LIN {X 0,Y 486.099,Z 588.304,A -85,B 0,C 180,E1 16517.76,E2 16517.76} C_VEL
LIN {X 0,Y 480.059,Z 803.394,A -85,B 0,C 180,E1 16513.95,E2 16513.95} C_VEL
LIN {X 0,Y 477.626,Z 893.821,A -85,B 0,C 180,E1 16512.362,E2 16512.362} C_VEL
LIN {X 0,Y 476.267,Z 916.596,A -85,B 0,C 180,E1 16511.765,E2 16511.765} C_VEL
LIN {X 0,Y 474.605,Z 939.076,A -85,B 0,C 180,E1 16510.978,E2 16510.978} C_VEL
LIN {X 0,Y 472.622,Z 960.372,A -85,B 0,C 180,E1 16510.02,E2 16510.02} C_VEL
LIN {X 0,Y 470.211,Z 983.19,A -85,B 0,C 180,E1 16508.757,E2 16508.757} C_VEL
LIN {X 0,Y 467.909,Z 1002.932,A -85,B 0,C 180,E1 16507.441,E2 16507.441} C_VEL
LIN {X 0,Y 465.309,Z 1023.138,A -85,B 0,C 180,E1 16505.842,E2 16505.842} C_VEL
LIN {X 0,Y 462.74,Z 1041.912,A -85,B 0,C 180,E1 16504.113,E2 16504.113} C_VEL
LIN {X 0,Y 460.177,Z 1059.991,A -85,B 0,C 180,E1 16502.163,E2 16502.163} C_VEL
LIN {X 0,Y 457.846,Z 1076.424,A -85,B 0,C 180,E1 16500.141,E2 16500.141} C_VEL
LIN {X 0,Y 455.797,Z 1090.318,A -85,B 0,C 180,E1 16498.135,E2 16498.135} C_VEL
LIN {X 0,Y 453.704,Z 1104.729,A -85,B 0,C 180,E1 16495.731,E2 16495.731} C_VEL
LIN {X 0,Y 451.938,Z 1117.804,A -85,B 0,C 180,E1 16493.192,E2 16493.192} C_VEL
LIN {X 0,Y 450.527,Z 1129.746,A -85,B 0,C 180,E1 16490.522,E2 16490.522} C_VEL
LIN {X 0,Y 449.445,Z 1140.142,A -85,B 0,C 180,E1 16487.745,E2 16487.745} C_VEL
LIN {X 0,Y 448.703,Z 1149.284,A -85,B 0,C 180,E1 16484.848,E2 16484.848} C_VEL
LIN {X 0,Y 448.284,Z 1155.954,A -85,B 0,C 180,E1 16482.233,E2 16482.233} C_VEL
LIN {X 0,Y 448.045,Z 1161.809,A -85,B 0,C 180,E1 16479.376,E2 16479.376} C_VEL
LIN {X 0,Y 447.94,Z 1165.827,A -85,B 0,C 180,E1 16476.643,E2 16476.643} C_VEL
LIN {X 0,Y 447.906,Z 1168.675,A -85,B 0,C 180,E1 16473.778,E2 16473.778} C_VEL
LIN {X 0,Y 447.893,Z 1169.826,A -85,B 0,C 180,E1 16471.023,E2 16471.023} C_VEL
LIN {X 0,Y 447.906,Z 1169.735,A -85,B 0,C 180,E1 16468.465,E2 16468.465} C_VEL
LIN {X 0,Y 447.911,Z 1168.068,A -85,B 0,C 180,E1 16465.519,E2 16465.519} C_VEL
LIN {X 0,Y 447.931,Z 1165.32,A -85,B 0,C 180,E1 16462.948,E2 16462.948} C_VEL
LIN {X 0,Y 448.063,Z 1160.59,A -85,B 0,C 180,E1 16459.976,E2 16459.976} C_VEL
LIN {X 0,Y 448.324,Z 1155.044,A -85,B 0,C 180,E1 16457.375,E2 16457.375} C_VEL
LIN {X 0,Y 448.874,Z 1146.956,A -85,B 0,C 180,E1 16454.364,E2 16454.364} C_VEL
LIN {X 0,Y 449.631,Z 1138.281,A -85,B 0,C 180,E1 16451.718,E2 16451.718} C_VEL
LIN {X 0,Y 450.833,Z 1126.863,A -85,B 0,C 180,E1 16448.807,E2 16448.807} C_VEL
LIN {X 0,Y 452.366,Z 1114.623,A -85,B 0,C 180,E1 16446.141,E2 16446.141} C_VEL
LIN {X 0,Y 454.239,Z 1100.876,A -85,B 0,C 180,E1 16443.6,E2 16443.6} C_VEL
LIN {X 0,Y 456.476,Z 1085.886,A -85,B 0,C 180,E1 16441.181,E2 16441.181} C_VEL
LIN {X 0,Y 458.665,Z 1070.559,A -85,B 0,C 180,E1 16439.111,E2 16439.111} C_VEL
LIN {X 0,Y 461.277,Z 1052.244,A -85,B 0,C 180,E1 16436.965,E2 16436.965} C_VEL
LIN {X 0,Y 463.797,Z 1034.322,A -85,B 0,C 180,E1 16435.16,E2 16435.16} C_VEL
LIN {X 0,Y 466.455,Z 1014.276,A -85,B 0,C 180,E1 16433.423,E2 16433.423} C_VEL
LIN {X 0,Y 468.782,Z 995.661,A -85,B 0,C 180,E1 16432.047,E2 16432.047} C_VEL
LIN {X 0,Y 471.222,Z 974.145,A -85,B 0,C 180,E1 16430.714,E2 16430.714} C_VEL
LIN {X 0,Y 473.181,Z 954.857,A -85,B 0,C 180,E1 16429.712,E2 16429.712} C_VEL
LIN {X 0,Y 475.154,Z 931.581,A -85,B 0,C 180,E1 16428.737,E2 16428.737} C_VEL
LIN {X 0,Y 476.803,Z 908.574,A -85,B 0,C 180,E1 16427.994,E2 16427.994} C_VEL
LIN {X 0,Y 477.948,Z 885.319,A -85,B 0,C 180,E1 16427.475,E2 16427.475} C_VEL
LIN {X 0,Y 483.619,Z 675.24,A -85,B 0,C 180,E1 16423.788,E2 16423.788} C_VEL
LIN {X 0,Y 486.084,Z 586.059,A -85,B 0,C 180,E1 16422.19,E2 16422.19} C_VEL
LIN {X 0,Y 473.889,Z 567.57,A -85,B 0,C 180,E1 16420.272,E2 16420.272} C_VEL
LIN {X 0,Y 464.24,Z 553.896,A -85,B 0,C 180,E1 16418.651,E2 16418.651} C_VEL
LIN {X 0,Y 460.411,Z 548.485,A -85,B 0,C 180,E1 16417.921,E2 16417.921} C_VEL
LIN {X 0,Y 456.172,Z 540.578,A -85,B 0,C 180,E1 16416.44,E2 16416.44} C_VEL
LIN {X 0,Y 453.762,Z 536.177,A -85,B 0,C 180,E1 16415.571,E2 16415.571} C_VEL
LIN {X 0,Y 451.433,Z 531.823,A -85,B 0,C 180,E1 16414.695,E2 16414.695} C_VEL
LIN {X 0,Y 449.419,Z 528.438,A -85,B 0,C 180,E1 16413.946,E2 16413.946} C_VEL
LIN {X 0,Y 449.153,Z 527.264,A -85,B 0,C 180,E1 16413.637,E2 16413.637} C_VEL
LIN {X 0,Y 449.125,Z 527.104,A -85,B 0,C 180,E1 16410.002,E2 16410.002} C_VEL
LIN {X 0,Y 449.124,Z 527.069,A -85,B 0,C 180,E1 16406.21,E2 16406.21} C_VEL
LIN {X 0,Y 449.124,Z 527.062,A -85,B 0,C 180,E1 16402.498,E2 16402.498} C_VEL
LIN {X 0,Y 449.126,Z 527.105,A -85,B 0,C 180,E1 16398.697,E2 16398.697} C_VEL
LIN {X 0,Y 449.13,Z 527.051,A -85,B 0,C 180,E1 16394.944,E2 16394.944} C_VEL
LIN {X 0,Y 449.124,Z 527.093,A -85,B 0,C 180,E1 16391.167,E2 16391.167} C_VEL
LIN {X 0,Y 449.134,Z 527.06,A -85,B 0,C 180,E1 16387.418,E2 16387.418} C_VEL
LIN {X 0,Y 449.12,Z 527.09,A -85,B 0,C 180,E1 16383.701,E2 16383.701} C_VEL
LIN {X 0,Y 449.134,Z 527.091,A -85,B 0,C 180,E1 16380,E2 16380} C_VEL
LIN {X 0,Y 449.126,Z 527.091,A -85,B 0,C 180,E1 16376.298,E2 16376.298} C_VEL
LIN {X 0,Y 449.14,Z 527.086,A -85,B 0,C 180,E1 16372.581,E2 16372.581} C_VEL
LIN {X 0,Y 449.116,Z 527.07,A -85,B 0,C 180,E1 16368.832,E2 16368.832} C_VEL
LIN {X 0,Y 449.124,Z 527.09,A -85,B 0,C 180,E1 16365.034,E2 16365.034} C_VEL
LIN {X 0,Y 449.127,Z 527.056,A -85,B 0,C 180,E1 16361.302,E2 16361.302} C_VEL
LIN {X 0,Y 449.133,Z 527.103,A -85,B 0,C 180,E1 16357.486,E2 16357.486} C_VEL
LIN {X 0,Y 449.123,Z 527.064,A -85,B 0,C 180,E1 16353.703,E2 16353.703} C_VEL
LIN {X 0,Y 449.114,Z 527.068,A -85,B 0,C 180,E1 16350.001,E2 16350.001} C_VEL
LIN {X 0,Y 449.131,Z 527.101,A -85,B 0,C 180,E1 16346.335,E2 16346.335} C_VEL
LIN {X 0,Y 449.156,Z 527.348,A -85,B 0,C 180,E1 16343.88,E2 16343.88} C_VEL
LIN {X 0,Y 450.468,Z 530.617,A -85,B 0,C 180,E1 16343.18,E2 16343.18} C_VEL
LIN {X 0,Y 451.904,Z 532.719,A -85,B 0,C 180,E1 16342.682,E2 16342.682} C_VEL
LIN {X 0,Y 453.881,Z 536.431,A -85,B 0,C 180,E1 16341.916,E2 16341.916} C_VEL
LIN {X 0,Y 459.677,Z 547.518,A -85,B 0,C 180,E1 16339.758,E2 16339.758} C_VEL
LIN {X 0,Y 466.824,Z 561.751,A -85,B 0,C 180,E1 16337.237,E2 16337.237} C_VEL
LIN {X 0,Y 474.929,Z 579.421,A -85,B 0,C 180,E1 16334.464,E2 16334.464} C_VEL
LIN {X 0,Y 476.317,Z 582.673,A -85,B 0,C 180,E1 16333.991,E2 16333.991} C_VEL
LIN {X 0,Y 476.279,Z 586.145,A -85,B 0,C 180,E1 16333.755,E2 16333.755} C_VEL
LIN {X 0,Y 481.634,Z 620.657,A -85,B 0,C 180,E1 16332.398,E2 16332.398} C_VEL
LIN {X 0,Y 478.079,Z 773.465,A -85,B 0,C 180,E1 16329.858,E2 16329.858} C_VEL
LIN {X 0,Y 477.186,Z 781.171,A -85,B 0,C 180,E1 16329.811,E2 16329.811} C_VEL
LIN {X 0,Y 472.133,Z 801.764,A -85,B 0,C 180,E1 16329.986,E2 16329.986} C_VEL
LIN {X 0,Y 471.436,Z 808.376,A -85,B 0,C 180,E1 16329.938,E2 16329.938} C_VEL
LIN {X 0,Y 469.256,Z 897.27,A -85,B 0,C 180,E1 16328.444,E2 16328.444} C_VEL
LIN {X 0,Y 467.96,Z 918.23,A -85,B 0,C 180,E1 16327.895,E2 16327.895} C_VEL
LIN {X 0,Y 466.239,Z 939.238,A -85,B 0,C 180,E1 16327.134,E2 16327.134} C_VEL
LIN {X 0,Y 464.225,Z 958.156,A -85,B 0,C 180,E1 16326.244,E2 16326.244} C_VEL
LIN {X 0,Y 461.634,Z 978.719,A -85,B 0,C 180,E1 16325.027,E2 16325.027} C_VEL
LIN {X 0,Y 458.991,Z 997.401,A -85,B 0,C 180,E1 16323.68,E2 16323.68} C_VEL
LIN {X 0,Y 456.137,Z 1015.398,A -85,B 0,C 180,E1 16322.111,E2 16322.111} C_VEL
LIN {X 0,Y 453.093,Z 1033.822,A -85,B 0,C 180,E1 16320.208,E2 16320.208} C_VEL
LIN {X 0,Y 450.29,Z 1050.571,A -85,B 0,C 180,E1 16318.172,E2 16318.172} C_VEL
LIN {X 0,Y 447.738,Z 1066.039,A -85,B 0,C 180,E1 16315.957,E2 16315.957} C_VEL
LIN {X 0,Y 445.461,Z 1080.363,A -85,B 0,C 180,E1 16313.549,E2 16313.549} C_VEL
LIN {X 0,Y 443.517,Z 1093.953,A -85,B 0,C 180,E1 16310.867,E2 16310.867} C_VEL
LIN {X 0,Y 442.1,Z 1105.41,A -85,B 0,C 180,E1 16308.186,E2 16308.186} C_VEL
LIN {X 0,Y 441.122,Z 1114.888,A -85,B 0,C 180,E1 16305.513,E2 16305.513} C_VEL
LIN {X 0,Y 440.486,Z 1123.199,A -85,B 0,C 180,E1 16302.72,E2 16302.72} C_VEL
LIN {X 0,Y 440.142,Z 1129.541,A -85,B 0,C 180,E1 16300.074,E2 16300.074} C_VEL
LIN {X 0,Y 439.969,Z 1134.242,A -85,B 0,C 180,E1 16297.443,E2 16297.443} C_VEL
LIN {X 0,Y 439.914,Z 1137.79,A -85,B 0,C 180,E1 16294.563,E2 16294.563} C_VEL
LIN {X 0,Y 439.902,Z 1139.558,A -85,B 0,C 180,E1 16291.954,E2 16291.954} C_VEL
LIN {X 0,Y 439.896,Z 1139.876,A -85,B 0,C 180,E1 16289.219,E2 16289.219} C_VEL
LIN {X 0,Y 439.91,Z 1138.777,A -85,B 0,C 180,E1 16286.482,E2 16286.482} C_VEL
LIN {X 0,Y 439.949,Z 1136.016,A -85,B 0,C 180,E1 16283.737,E2 16283.737} C_VEL
LIN {X 0,Y 440.075,Z 1131.495,A -85,B 0,C 180,E1 16280.849,E2 16280.849} C_VEL
LIN {X 0,Y 440.352,Z 1125.545,A -85,B 0,C 180,E1 16278.075,E2 16278.075} C_VEL
LIN {X 0,Y 440.843,Z 1118.111,A -85,B 0,C 180,E1 16275.419,E2 16275.419} C_VEL
LIN {X 0,Y 441.776,Z 1108.232,A -85,B 0,C 180,E1 16272.481,E2 16272.481} C_VEL
LIN {X 0,Y 443.044,Z 1097.668,A -85,B 0,C 180,E1 16269.856,E2 16269.856} C_VEL
LIN {X 0,Y 444.652,Z 1085.845,A -85,B 0,C 180,E1 16267.386,E2 16267.386} C_VEL
LIN {X 0,Y 446.704,Z 1072.366,A -85,B 0,C 180,E1 16264.973,E2 16264.973} C_VEL
LIN {X 0,Y 449.123,Z 1057.615,A -85,B 0,C 180,E1 16262.703,E2 16262.703} C_VEL
LIN {X 0,Y 451.767,Z 1041.722,A -85,B 0,C 180,E1 16260.621,E2 16260.621} C_VEL
LIN {X 0,Y 454.601,Z 1024.814,A -85,B 0,C 180,E1 16258.73,E2 16258.73} C_VEL
LIN {X 0,Y 457.503,Z 1007.003,A -85,B 0,C 180,E1 16257.031,E2 16257.031} C_VEL
LIN {X 0,Y 460.175,Z 989.112,A -85,B 0,C 180,E1 16255.603,E2 16255.603} C_VEL
LIN {X 0,Y 462.828,Z 969.742,A -85,B 0,C 180,E1 16254.318,E2 16254.318} C_VEL
LIN {X 0,Y 465.075,Z 950.87,A -85,B 0,C 180,E1 16253.297,E2 16253.297} C_VEL
LIN {X 0,Y 467.035,Z 929.824,A -85,B 0,C 180,E1 16252.405,E2 16252.405} C_VEL
LIN {X 0,Y 468.671,Z 907.781,A -85,B 0,C 180,E1 16251.717,E2 16251.717} C_VEL
LIN {X 0,Y 469.662,Z 886.494,A -85,B 0,C 180,E1 16251.264,E2 16251.264} C_VEL
LIN {X 0,Y 475.072,Z 656.342,A -85,B 0,C 180,E1 16247.434,E2 16247.434} C_VEL
LIN {X 0,Y 475.695,Z 625.368,A -85,B 0,C 180,E1 16246.882,E2 16246.882} C_VEL
LIN {X 0,Y 468.087,Z 586.907,A -85,B 0,C 180,E1 16245.103,E2 16245.103} C_VEL
LIN {X 0,Y 466.861,Z 584.352,A -85,B 0,C 180,E1 16244.798,E2 16244.798} C_VEL
LIN {X 0,Y 459.918,Z 567.603,A -85,B 0,C 180,E1 16241.868,E2 16241.868} C_VEL
LIN {X 0,Y 454.611,Z 555.916,A -85,B 0,C 180,E1 16239.589,E2 16239.589} C_VEL
LIN {X 0,Y 451.777,Z 555.588,A -85,B 0,C 180,E1 16239.029,E2 16239.029} C_VEL
LIN {X 0,Y 451.766,Z 556.321,A -85,B 0,C 180,E1 16238.826,E2 16238.826} C_VEL
LIN {X 0,Y 455.537,Z 567.842,A -85,B 0,C 180,E1 16237.5,E2 16237.5} C_VEL
LIN {X 0,Y 453.889,Z 610.869,A -85,B 0,C 180,E1 16233.851,E2 16233.851} C_VEL
LIN {X 0,Y 452.299,Z 651.564,A -85,B 0,C 180,E1 16230.413,E2 16230.413} C_VEL
LIN {X 0,Y 450.385,Z 696.261,A -85,B 0,C 180,E1 16226.644,E2 16226.644} C_VEL
LIN {X 0,Y 449.613,Z 717.199,A -85,B 0,C 180,E1 16224.91,E2 16224.91} C_VEL
LIN {X 0,Y 450.51,Z 726.614,A -85,B 0,C 180,E1 16224.68,E2 16224.68} C_VEL
LIN {X 0,Y 447.879,Z 888.58,A -85,B 0,C 180,E1 16221.821,E2 16221.821} C_VEL
LIN {X 0,Y 447.488,Z 906.098,A -85,B 0,C 180,E1 16221.269,E2 16221.269} C_VEL
LIN {X 0,Y 446.873,Z 922.97,A -85,B 0,C 180,E1 16220.498,E2 16220.498} C_VEL
LIN {X 0,Y 446.129,Z 939.205,A -85,B 0,C 180,E1 16219.508,E2 16219.508} C_VEL
LIN {X 0,Y 445.263,Z 954.342,A -85,B 0,C 180,E1 16218.324,E2 16218.324} C_VEL
LIN {X 0,Y 444.373,Z 968.446,A -85,B 0,C 180,E1 16216.941,E2 16216.941} C_VEL
LIN {X 0,Y 443.488,Z 981.556,A -85,B 0,C 180,E1 16215.362,E2 16215.362} C_VEL
LIN {X 0,Y 442.721,Z 992.693,A -85,B 0,C 180,E1 16213.718,E2 16213.718} C_VEL
LIN {X 0,Y 442.045,Z 1002.767,A -85,B 0,C 180,E1 16211.879,E2 16211.879} C_VEL
LIN {X 0,Y 441.514,Z 1011.448,A -85,B 0,C 180,E1 16209.899,E2 16209.899} C_VEL
LIN {X 0,Y 441.138,Z 1018.585,A -85,B 0,C 180,E1 16207.816,E2 16207.816} C_VEL
LIN {X 0,Y 440.923,Z 1023.899,A -85,B 0,C 180,E1 16205.727,E2 16205.727} C_VEL
LIN {X 0,Y 440.814,Z 1027.687,A -85,B 0,C 180,E1 16203.511,E2 16203.511} C_VEL
LIN {X 0,Y 440.796,Z 1029.775,A -85,B 0,C 180,E1 16201.3,E2 16201.3} C_VEL
LIN {X 0,Y 440.842,Z 1030.214,A -85,B 0,C 180,E1 16199.091,E2 16199.091} C_VEL
LIN {X 0,Y 440.91,Z 1028.924,A -85,B 0,C 180,E1 16196.88,E2 16196.88} C_VEL
LIN {X 0,Y 441.068,Z 1025.904,A -85,B 0,C 180,E1 16194.667,E2 16194.667} C_VEL
LIN {X 0,Y 441.357,Z 1021.069,A -85,B 0,C 180,E1 16192.45,E2 16192.45} C_VEL
LIN {X 0,Y 441.775,Z 1014.603,A -85,B 0,C 180,E1 16190.359,E2 16190.359} C_VEL
LIN {X 0,Y 442.316,Z 1006.606,A -85,B 0,C 180,E1 16188.394,E2 16188.394} C_VEL
LIN {X 0,Y 442.981,Z 997.146,A -85,B 0,C 180,E1 16186.557,E2 16186.557} C_VEL
LIN {X 0,Y 443.747,Z 986.173,A -85,B 0,C 180,E1 16184.849,E2 16184.849} C_VEL
LIN {X 0,Y 444.574,Z 973.502,A -85,B 0,C 180,E1 16183.27,E2 16183.27} C_VEL
LIN {X 0,Y 445.376,Z 959.71,A -85,B 0,C 180,E1 16181.885,E2 16181.885} C_VEL
LIN {X 0,Y 446.045,Z 945.712,A -85,B 0,C 180,E1 16180.761,E2 16180.761} C_VEL
LIN {X 0,Y 446.633,Z 930.284,A -85,B 0,C 180,E1 16179.796,E2 16179.796} C_VEL
LIN {X 0,Y 447.099,Z 912.684,A -85,B 0,C 180,E1 16178.979,E2 16178.979} C_VEL
LIN {X 0,Y 447.333,Z 895.443,A -85,B 0,C 180,E1 16178.434,E2 16178.434} C_VEL
LIN {X 0,Y 449.136,Z 771.991,A -85,B 0,C 180,E1 16176.209,E2 16176.209} C_VEL
LIN {X 0,Y 450.268,Z 727.667,A -85,B 0,C 180,E1 16175.325,E2 16175.325} C_VEL
LIN {X 0,Y 450.922,Z 722.428,A -85,B 0,C 180,E1 16174.944,E2 16174.944} C_VEL
LIN {X 0,Y 452.009,Z 681.094,A -85,B 0,C 180,E1 16171.69,E2 16171.69} C_VEL
LIN {X 0,Y 452.655,Z 642.043,A -85,B 0,C 180,E1 16168.73,E2 16168.73} C_VEL
LIN {X 0,Y 452.801,Z 603.805,A -85,B 0,C 180,E1 16165.953,E2 16165.953} C_VEL
LIN {X 0,Y 452.703,Z 562.114,A -85,B 0,C 180,E1 16163.037,E2 16163.037} C_VEL
LIN {X 0,Y 453.595,Z 560.379,A -85,B 0,C 180,E1 16162.766,E2 16162.766} C_VEL
LIN {X 0,Y 456.982,Z 558.136,A -85,B 0,C 180,E1 16162.3,E2 16162.3} C_VEL
LIN {X 0,Y 457.592,Z 557.709,A -85,B 0,C 180,E1 16162.22,E2 16162.22} C_VEL
LIN {X 0,Y 469.198,Z 574.103,A -85,B 0,C 180,E1 16160.201,E2 16160.201} C_VEL
LIN {X 0,Y 480.371,Z 591.263,A -85,B 0,C 180,E1 16158.387,E2 16158.387} C_VEL
LIN {X 0,Y 474.097,Z 800.438,A -85,B 0,C 180,E1 16154.635,E2 16154.635} C_VEL
LIN {X 0,Y 471.323,Z 893.219,A -85,B 0,C 180,E1 16152.97,E2 16152.97} C_VEL
LIN {X 0,Y 469.85,Z 916.411,A -85,B 0,C 180,E1 16152.355,E2 16152.355} C_VEL
LIN {X 0,Y 468.07,Z 939.12,A -85,B 0,C 180,E1 16151.55,E2 16151.55} C_VEL
LIN {X 0,Y 466.092,Z 959.379,A -85,B 0,C 180,E1 16150.629,E2 16150.629} C_VEL
LIN {X 0,Y 463.687,Z 981.141,A -85,B 0,C 180,E1 16149.431,E2 16149.431} C_VEL
LIN {X 0,Y 461.218,Z 1001.087,A -85,B 0,C 180,E1 16148.101,E2 16148.101} C_VEL
LIN {X 0,Y 458.352,Z 1022.674,A -85,B 0,C 180,E1 16146.395,E2 16146.395} C_VEL
LIN {X 0,Y 455.838,Z 1040.251,A -85,B 0,C 180,E1 16144.771,E2 16144.771} C_VEL
LIN {X 0,Y 453.017,Z 1059.1,A -85,B 0,C 180,E1 16142.734,E2 16142.734} C_VEL
LIN {X 0,Y 450.477,Z 1076.063,A -85,B 0,C 180,E1 16140.623,E2 16140.623} C_VEL
LIN {X 0,Y 448.125,Z 1091.56,A -85,B 0,C 180,E1 16138.376,E2 16138.376} C_VEL
LIN {X 0,Y 446.209,Z 1104.727,A -85,B 0,C 180,E1 16136.196,E2 16136.196} C_VEL
LIN {X 0,Y 444.297,Z 1117.802,A -85,B 0,C 180,E1 16133.614,E2 16133.614} C_VEL
LIN {X 0,Y 442.769,Z 1129.721,A -85,B 0,C 180,E1 16130.904,E2 16130.904} C_VEL
LIN {X 0,Y 441.594,Z 1140.141,A -85,B 0,C 180,E1 16128.071,E2 16128.071} C_VEL
LIN {X 0,Y 440.785,Z 1149.285,A -85,B 0,C 180,E1 16125.121,E2 16125.121} C_VEL
LIN {X 0,Y 440.319,Z 1155.954,A -85,B 0,C 180,E1 16122.458,E2 16122.458} C_VEL
LIN {X 0,Y 440.051,Z 1161.809,A -85,B 0,C 180,E1 16119.548,E2 16119.548} C_VEL
LIN {X 0,Y 439.937,Z 1165.799,A -85,B 0,C 180,E1 16116.787,E2 16116.787} C_VEL
LIN {X 0,Y 439.91,Z 1168.632,A -85,B 0,C 180,E1 16113.91,E2 16113.91} C_VEL
LIN {X 0,Y 439.894,Z 1169.826,A -85,B 0,C 180,E1 16111.042,E2 16111.042} C_VEL
LIN {X 0,Y 439.906,Z 1169.735,A -85,B 0,C 180,E1 16108.437,E2 16108.437} C_VEL
LIN {X 0,Y 439.911,Z 1168.068,A -85,B 0,C 180,E1 16105.437,E2 16105.437} C_VEL
LIN {X 0,Y 439.934,Z 1165.319,A -85,B 0,C 180,E1 16102.819,E2 16102.819} C_VEL
LIN {X 0,Y 440.086,Z 1160.59,A -85,B 0,C 180,E1 16099.793,E2 16099.793} C_VEL
LIN {X 0,Y 440.37,Z 1155.044,A -85,B 0,C 180,E1 16097.144,E2 16097.144} C_VEL
LIN {X 0,Y 440.989,Z 1146.767,A -85,B 0,C 180,E1 16094.014,E2 16094.014} C_VEL
LIN {X 0,Y 441.849,Z 1137.851,A -85,B 0,C 180,E1 16091.256,E2 16091.256} C_VEL
LIN {X 0,Y 443.134,Z 1126.662,A -85,B 0,C 180,E1 16088.373,E2 16088.373} C_VEL
LIN {X 0,Y 444.765,Z 1114.625,A -85,B 0,C 180,E1 16085.707,E2 16085.707} C_VEL
LIN {X 0,Y 446.661,Z 1101.614,A -85,B 0,C 180,E1 16083.26,E2 16083.26} C_VEL
LIN {X 0,Y 448.938,Z 1086.274,A -85,B 0,C 180,E1 16080.814,E2 16080.814} C_VEL
LIN {X 0,Y 451.325,Z 1070.265,A -85,B 0,C 180,E1 16078.626,E2 16078.626} C_VEL
LIN {X 0,Y 454.106,Z 1051.924,A -85,B 0,C 180,E1 16076.45,E2 16076.45} C_VEL
LIN {X 0,Y 456.656,Z 1034.666,A -85,B 0,C 180,E1 16074.687,E2 16074.687} C_VEL
LIN {X 0,Y 459.555,Z 1013.715,A -85,B 0,C 180,E1 16072.86,E2 16072.86} C_VEL
LIN {X 0,Y 462.317,Z 992.834,A -85,B 0,C 180,E1 16071.316,E2 16071.316} C_VEL
LIN {X 0,Y 464.727,Z 972.039,A -85,B 0,C 180,E1 16070.042,E2 16070.042} C_VEL
LIN {X 0,Y 466.98,Z 950.663,A -85,B 0,C 180,E1 16068.944,E2 16068.944} C_VEL
LIN {X 0,Y 468.95,Z 928.17,A -85,B 0,C 180,E1 16068.034,E2 16068.034} C_VEL
LIN {X 0,Y 470.708,Z 903.822,A -85,B 0,C 180,E1 16067.288,E2 16067.288} C_VEL
LIN {X 0,Y 471.826,Z 881.099,A -85,B 0,C 180,E1 16066.792,E2 16066.792} C_VEL
LIN {X 0,Y 478.044,Z 668.473,A -85,B 0,C 180,E1 16063.004,E2 16063.004} C_VEL
LIN {X 0,Y 480.314,Z 589.595,A -85,B 0,C 180,E1 16061.569,E2 16061.569} C_VEL
LIN {X 0,Y 467.768,Z 570.524,A -85,B 0,C 180,E1 16059.527,E2 16059.527} C_VEL
LIN {X 0,Y 456.907,Z 555.345,A -85,B 0,C 180,E1 16057.628,E2 16057.628} C_VEL
LIN {X 0,Y 452.567,Z 549.341,A -85,B 0,C 180,E1 16056.778,E2 16056.778} C_VEL
LIN {X 0,Y 448.633,Z 542.069,A -85,B 0,C 180,E1 16055.343,E2 16055.343} C_VEL
LIN {X 0,Y 446.098,Z 537.508,A -85,B 0,C 180,E1 16054.389,E2 16054.389} C_VEL
LIN {X 0,Y 444.034,Z 533.552,A -85,B 0,C 180,E1 16053.559,E2 16053.559} C_VEL
LIN {X 0,Y 441.519,Z 529.538,A -85,B 0,C 180,E1 16052.602,E2 16052.602} C_VEL
LIN {X 0,Y 441.214,Z 528.299,A -85,B 0,C 180,E1 16052.298,E2 16052.298} C_VEL
LIN {X 0,Y 441.194,Z 528.061,A -85,B 0,C 180,E1 16048.712,E2 16048.712} C_VEL
LIN {X 0,Y 441.188,Z 528.088,A -85,B 0,C 180,E1 16044.931,E2 16044.931} C_VEL
LIN {X 0,Y 441.19,Z 528.043,A -85,B 0,C 180,E1 16041.12,E2 16041.12} C_VEL
LIN {X 0,Y 441.185,Z 528.072,A -85,B 0,C 180,E1 16037.406,E2 16037.406} C_VEL
LIN {X 0,Y 441.192,Z 528.06,A -85,B 0,C 180,E1 16033.632,E2 16033.632} C_VEL
LIN {X 0,Y 441.181,Z 528.049,A -85,B 0,C 180,E1 16029.918,E2 16029.918} C_VEL
LIN {X 0,Y 441.187,Z 528.079,A -85,B 0,C 180,E1 16026.114,E2 16026.114} C_VEL
LIN {X 0,Y 441.191,Z 528.084,A -85,B 0,C 180,E1 16022.338,E2 16022.338} C_VEL
LIN {X 0,Y 441.19,Z 528.087,A -85,B 0,C 180,E1 16018.571,E2 16018.571} C_VEL
LIN {X 0,Y 441.192,Z 528.089,A -85,B 0,C 180,E1 16014.799,E2 16014.799} C_VEL
LIN {X 0,Y 441.182,Z 528.094,A -85,B 0,C 180,E1 16011.135,E2 16011.135} C_VEL
LIN {X 0,Y 441.184,Z 528.037,A -85,B 0,C 180,E1 16007.301,E2 16007.301} C_VEL
LIN {X 0,Y 441.191,Z 528.089,A -85,B 0,C 180,E1 16003.543,E2 16003.543} C_VEL
LIN {X 0,Y 441.189,Z 528.048,A -85,B 0,C 180,E1 15999.712,E2 15999.712} C_VEL
LIN {X 0,Y 441.177,Z 528.062,A -85,B 0,C 180,E1 15996.066,E2 15996.066} C_VEL
LIN {X 0,Y 441.184,Z 528.086,A -85,B 0,C 180,E1 15992.316,E2 15992.316} C_VEL
LIN {X 0,Y 441.191,Z 528.047,A -85,B 0,C 180,E1 15988.584,E2 15988.584} C_VEL
LIN {X 0,Y 441.223,Z 528.339,A -85,B 0,C 180,E1 15985.255,E2 15985.255} C_VEL
LIN {X 0,Y 442.566,Z 531.64,A -85,B 0,C 180,E1 15984.505,E2 15984.505} C_VEL
LIN {X 0,Y 444.11,Z 534.001,A -85,B 0,C 180,E1 15983.925,E2 15983.925} C_VEL
LIN {X 0,Y 447.13,Z 539.687,A -85,B 0,C 180,E1 15982.699,E2 15982.699} C_VEL
LIN {X 0,Y 451.849,Z 548.388,A -85,B 0,C 180,E1 15980.901,E2 15980.901} C_VEL
LIN {X 0,Y 458.102,Z 560.665,A -85,B 0,C 180,E1 15978.598,E2 15978.598} C_VEL
LIN {X 0,Y 466.059,Z 577.61,A -85,B 0,C 180,E1 15975.77,E2 15975.77} C_VEL
LIN {X 0,Y 469.611,Z 585.346,A -85,B 0,C 180,E1 15974.634,E2 15974.634} C_VEL
LIN {X 0,Y 470.709,Z 587.684,A -85,B 0,C 180,E1 15974.44,E2 15974.44} C_VEL
LIN {X 0,Y 475.957,Z 622.19,A -85,B 0,C 180,E1 15973.055,E2 15973.055} C_VEL
LIN {X 0,Y 471.436,Z 808.376,A -85,B 0,C 180,E1 15969.938,E2 15969.938} C_VEL
LIN {X 0,Y 470.53,Z 816.08,A -85,B 0,C 180,E1 15969.893,E2 15969.893} C_VEL
LIN {X 0,Y 465.433,Z 836.659,A -85,B 0,C 180,E1 15970.076,E2 15970.076} C_VEL
LIN {X 0,Y 464.73,Z 843.27,A -85,B 0,C 180,E1 15970.029,E2 15970.029} C_VEL
LIN {X 0,Y 463.239,Z 898.428,A -85,B 0,C 180,E1 15969.079,E2 15969.079} C_VEL
LIN {X 0,Y 461.858,Z 919.433,A -85,B 0,C 180,E1 15968.516,E2 15968.516} C_VEL
LIN {X 0,Y 459.974,Z 940.901,A -85,B 0,C 180,E1 15967.72,E2 15967.72} C_VEL
LIN {X 0,Y 457.76,Z 960.867,A -85,B 0,C 180,E1 15966.761,E2 15966.761} C_VEL
LIN {X 0,Y 455.203,Z 980.095,A -85,B 0,C 180,E1 15965.597,E2 15965.597} C_VEL
LIN {X 0,Y 452.421,Z 998.847,A -85,B 0,C 180,E1 15964.226,E2 15964.226} C_VEL
LIN {X 0,Y 449.57,Z 1015.981,A -85,B 0,C 180,E1 15962.714,E2 15962.714} C_VEL
LIN {X 0,Y 446.421,Z 1033.773,A -85,B 0,C 180,E1 15960.857,E2 15960.857} C_VEL
LIN {X 0,Y 443.482,Z 1050.159,A -85,B 0,C 180,E1 15958.847,E2 15958.847} C_VEL
LIN {X 0,Y 440.7,Z 1065.445,A -85,B 0,C 180,E1 15956.631,E2 15956.631} C_VEL
LIN {X 0,Y 438.259,Z 1079.584,A -85,B 0,C 180,E1 15954.246,E2 15954.246} C_VEL
LIN {X 0,Y 436.197,Z 1092.683,A -85,B 0,C 180,E1 15951.657,E2 15951.657} C_VEL
LIN {X 0,Y 434.566,Z 1104.312,A -85,B 0,C 180,E1 15948.93,E2 15948.93} C_VEL
LIN {X 0,Y 433.419,Z 1113.995,A -85,B 0,C 180,E1 15946.209,E2 15946.209} C_VEL
LIN {X 0,Y 432.618,Z 1122.71,A -85,B 0,C 180,E1 15943.227,E2 15943.227} C_VEL
LIN {X 0,Y 432.191,Z 1129.301,A -85,B 0,C 180,E1 15940.396,E2 15940.396} C_VEL
LIN {X 0,Y 431.978,Z 1134.243,A -85,B 0,C 180,E1 15937.581,E2 15937.581} C_VEL
LIN {X 0,Y 431.913,Z 1137.791,A -85,B 0,C 180,E1 15934.647,E2 15934.647} C_VEL
LIN {X 0,Y 431.902,Z 1139.558,A -85,B 0,C 180,E1 15931.99,E2 15931.99} C_VEL
LIN {X 0,Y 431.897,Z 1139.875,A -85,B 0,C 180,E1 15929.204,E2 15929.204} C_VEL
LIN {X 0,Y 431.91,Z 1138.777,A -85,B 0,C 180,E1 15926.416,E2 15926.416} C_VEL
LIN {X 0,Y 431.954,Z 1136.014,A -85,B 0,C 180,E1 15923.621,E2 15923.621} C_VEL
LIN {X 0,Y 432.09,Z 1131.493,A -85,B 0,C 180,E1 15920.678,E2 15920.678} C_VEL
LIN {X 0,Y 432.423,Z 1125.342,A -85,B 0,C 180,E1 15917.718,E2 15917.718} C_VEL
LIN {X 0,Y 433.007,Z 1118.064,A -85,B 0,C 180,E1 15915.012,E2 15915.012} C_VEL
LIN {X 0,Y 434.009,Z 1108.692,A -85,B 0,C 180,E1 15912.157,E2 15912.157} C_VEL
LIN {X 0,Y 435.427,Z 1097.96,A -85,B 0,C 180,E1 15909.431,E2 15909.431} C_VEL
LIN {X 0,Y 437.284,Z 1085.643,A -85,B 0,C 180,E1 15906.807,E2 15906.807} C_VEL
LIN {X 0,Y 439.498,Z 1072.294,A -85,B 0,C 180,E1 15904.389,E2 15904.389} C_VEL
LIN {X 0,Y 442.214,Z 1057.04,A -85,B 0,C 180,E1 15902.02,E2 15902.02} C_VEL
LIN {X 0,Y 445.076,Z 1041.315,A -85,B 0,C 180,E1 15899.936,E2 15899.936} C_VEL
LIN {X 0,Y 448.046,Z 1024.717,A -85,B 0,C 180,E1 15898.069,E2 15898.069} C_VEL
LIN {X 0,Y 451.13,Z 1006.817,A -85,B 0,C 180,E1 15896.352,E2 15896.352} C_VEL
LIN {X 0,Y 453.827,Z 989.588,A -85,B 0,C 180,E1 15894.975,E2 15894.975} C_VEL
LIN {X 0,Y 456.588,Z 970.018,A -85,B 0,C 180,E1 15893.676,E2 15893.676} C_VEL
LIN {X 0,Y 458.93,Z 950.974,A -85,B 0,C 180,E1 15892.644,E2 15892.644} C_VEL
LIN {X 0,Y 460.97,Z 929.983,A -85,B 0,C 180,E1 15891.753,E2 15891.753} C_VEL
LIN {X 0,Y 462.678,Z 907.912,A -85,B 0,C 180,E1 15891.061,E2 15891.061} C_VEL
LIN {X 0,Y 463.713,Z 886.558,A -85,B 0,C 180,E1 15890.605,E2 15890.605} C_VEL
LIN {X 0,Y 469.454,Z 656.094,A -85,B 0,C 180,E1 15886.735,E2 15886.735} C_VEL
LIN {X 0,Y 470.084,Z 627.151,A -85,B 0,C 180,E1 15886.214,E2 15886.214} C_VEL
LIN {X 0,Y 463.096,Z 591.291,A -85,B 0,C 180,E1 15884.52,E2 15884.52} C_VEL
LIN {X 0,Y 458.74,Z 584.129,A -85,B 0,C 180,E1 15883.704,E2 15883.704} C_VEL
LIN {X 0,Y 451.637,Z 567.187,A -85,B 0,C 180,E1 15880.592,E2 15880.592} C_VEL
LIN {X 0,Y 449.335,Z 562.385,A -85,B 0,C 180,E1 15879.607,E2 15879.607} C_VEL
LIN {X 0,Y 445.942,Z 562.006,A -85,B 0,C 180,E1 15878.962,E2 15878.962} C_VEL
LIN {X 0,Y 445.946,Z 562.999,A -85,B 0,C 180,E1 15878.716,E2 15878.716} C_VEL
LIN {X 0,Y 448.408,Z 570.687,A -85,B 0,C 180,E1 15877.821,E2 15877.821} C_VEL
LIN {X 0,Y 446.684,Z 613.305,A -85,B 0,C 180,E1 15874.183,E2 15874.183} C_VEL
LIN {X 0,Y 444.968,Z 654.54,A -85,B 0,C 180,E1 15870.669,E2 15870.669} C_VEL
LIN {X 0,Y 443,Z 698.558,A -85,B 0,C 180,E1 15866.934,E2 15866.934} C_VEL
LIN {X 0,Y 442.273,Z 718.211,A -85,B 0,C 180,E1 15865.304,E2 15865.304} C_VEL
LIN {X 0,Y 443.15,Z 727.442,A -85,B 0,C 180,E1 15865.074,E2 15865.074} C_VEL
LIN {X 0,Y 440.309,Z 889.78,A -85,B 0,C 180,E1 15862.136,E2 15862.136} C_VEL
LIN {X 0,Y 439.9,Z 907.457,A -85,B 0,C 180,E1 15861.566,E2 15861.566} C_VEL
LIN {X 0,Y 439.228,Z 925.24,A -85,B 0,C 180,E1 15860.731,E2 15860.731} C_VEL
LIN {X 0,Y 438.459,Z 941.278,A -85,B 0,C 180,E1 15859.725,E2 15859.725} C_VEL
LIN {X 0,Y 437.545,Z 956.487,A -85,B 0,C 180,E1 15858.496,E2 15858.496} C_VEL
LIN {X 0,Y 436.603,Z 970.883,A -85,B 0,C 180,E1 15857.046,E2 15857.046} C_VEL
LIN {X 0,Y 435.693,Z 983.842,A -85,B 0,C 180,E1 15855.439,E2 15855.439} C_VEL
LIN {X 0,Y 434.864,Z 995.175,A -85,B 0,C 180,E1 15853.699,E2 15853.699} C_VEL
LIN {X 0,Y 434.138,Z 1005.713,A -85,B 0,C 180,E1 15851.694,E2 15851.694} C_VEL
LIN {X 0,Y 433.615,Z 1014.088,A -85,B 0,C 180,E1 15849.691,E2 15849.691} C_VEL
LIN {X 0,Y 433.236,Z 1020.932,A -85,B 0,C 180,E1 15847.559,E2 15847.559} C_VEL
LIN {X 0,Y 433.017,Z 1026.24,A -85,B 0,C 180,E1 15845.3,E2 15845.3} C_VEL
LIN {X 0,Y 432.935,Z 1029.733,A -85,B 0,C 180,E1 15843.045,E2 15843.045} C_VEL
LIN {X 0,Y 432.93,Z 1031.452,A -85,B 0,C 180,E1 15840.794,E2 15840.794} C_VEL
LIN {X 0,Y 432.979,Z 1031.485,A -85,B 0,C 180,E1 15838.545,E2 15838.545} C_VEL
LIN {X 0,Y 433.089,Z 1029.841,A -85,B 0,C 180,E1 15836.294,E2 15836.294} C_VEL
LIN {X 0,Y 433.304,Z 1026.447,A -85,B 0,C 180,E1 15834.04,E2 15834.04} C_VEL
LIN {X 0,Y 433.621,Z 1021.457,A -85,B 0,C 180,E1 15831.915,E2 15831.915} C_VEL
LIN {X 0,Y 434.115,Z 1014.583,A -85,B 0,C 180,E1 15829.785,E2 15829.785} C_VEL
LIN {X 0,Y 434.736,Z 1006.172,A -85,B 0,C 180,E1 15827.785,E2 15827.785} C_VEL
LIN {X 0,Y 435.475,Z 996.128,A -85,B 0,C 180,E1 15825.914,E2 15825.914} C_VEL
LIN {X 0,Y 436.325,Z 984.459,A -85,B 0,C 180,E1 15824.176,E2 15824.176} C_VEL
LIN {X 0,Y 437.189,Z 971.606,A -85,B 0,C 180,E1 15822.636,E2 15822.636} C_VEL
LIN {X 0,Y 437.97,Z 957.618,A -85,B 0,C 180,E1 15821.299,E2 15821.299} C_VEL
LIN {X 0,Y 438.691,Z 942.447,A -85,B 0,C 180,E1 15820.148,E2 15820.148} C_VEL
LIN {X 0,Y 439.249,Z 926.894,A -85,B 0,C 180,E1 15819.236,E2 15819.236} C_VEL
LIN {X 0,Y 439.632,Z 909.779,A -85,B 0,C 180,E1 15818.509,E2 15818.509} C_VEL
LIN {X 0,Y 439.793,Z 891.745,A -85,B 0,C 180,E1 15818.004,E2 15818.004} C_VEL
LIN {X 0,Y 441.474,Z 786.272,A -85,B 0,C 180,E1 15816.069,E2 15816.069} C_VEL
LIN {X 0,Y 442.993,Z 730.018,A -85,B 0,C 180,E1 15814.928,E2 15814.928} C_VEL
LIN {X 0,Y 443.809,Z 725.336,A -85,B 0,C 180,E1 15814.611,E2 15814.611} C_VEL
LIN {X 0,Y 444.991,Z 684.953,A -85,B 0,C 180,E1 15811.407,E2 15811.407} C_VEL
LIN {X 0,Y 445.741,Z 644.804,A -85,B 0,C 180,E1 15808.339,E2 15808.339} C_VEL
LIN {X 0,Y 446.014,Z 606.611,A -85,B 0,C 180,E1 15805.533,E2 15805.533} C_VEL
LIN {X 0,Y 446.144,Z 579.868,A -85,B 0,C 180,E1 15803.607,E2 15803.607} C_VEL
LIN {X 0,Y 447.04,Z 578.05,A -85,B 0,C 180,E1 15803.333,E2 15803.333} C_VEL
LIN {X 0,Y 449.82,Z 575.94,A -85,B 0,C 180,E1 15802.938,E2 15802.938} C_VEL
LIN {X 0,Y 453.373,Z 570.82,A -85,B 0,C 180,E1 15802.526,E2 15802.526} C_VEL
LIN {X 0,Y 455.061,Z 567.651,A -85,B 0,C 180,E1 15802.352,E2 15802.352} C_VEL
LIN {X 0,Y 456.237,Z 567.211,A -85,B 0,C 180,E1 15802.188,E2 15802.188} C_VEL
LIN {X 0,Y 470.309,Z 587.94,A -85,B 0,C 180,E1 15799.738,E2 15799.738} C_VEL
LIN {X 0,Y 474.689,Z 595.261,A -85,B 0,C 180,E1 15799.008,E2 15799.008} C_VEL
LIN {X 0,Y 467.871,Z 809.184,A -85,B 0,C 180,E1 15795.132,E2 15795.132} C_VEL
LIN {X 0,Y 465.162,Z 893.135,A -85,B 0,C 180,E1 15793.6,E2 15793.6} C_VEL
LIN {X 0,Y 463.597,Z 916.035,A -85,B 0,C 180,E1 15792.984,E2 15792.984} C_VEL
LIN {X 0,Y 461.692,Z 938.577,A -85,B 0,C 180,E1 15792.172,E2 15792.172} C_VEL
LIN {X 0,Y 459.494,Z 959.564,A -85,B 0,C 180,E1 15791.199,E2 15791.199} C_VEL
LIN {X 0,Y 456.902,Z 981.62,A -85,B 0,C 180,E1 15789.962,E2 15789.962} C_VEL
LIN {X 0,Y 454.321,Z 1001.399,A -85,B 0,C 180,E1 15788.623,E2 15788.623} C_VEL
LIN {X 0,Y 451.292,Z 1022.976,A -85,B 0,C 180,E1 15786.889,E2 15786.889} C_VEL
LIN {X 0,Y 448.468,Z 1041.852,A -85,B 0,C 180,E1 15785.115,E2 15785.115} C_VEL
LIN {X 0,Y 445.627,Z 1059.953,A -85,B 0,C 180,E1 15783.117,E2 15783.117} C_VEL
LIN {X 0,Y 442.904,Z 1077.132,A -85,B 0,C 180,E1 15780.925,E2 15780.925} C_VEL
LIN {X 0,Y 440.425,Z 1092.605,A -85,B 0,C 180,E1 15778.621,E2 15778.621} C_VEL
LIN {X 0,Y 438.094,Z 1107.937,A -85,B 0,C 180,E1 15775.989,E2 15775.989} C_VEL
LIN {X 0,Y 436.405,Z 1119.704,A -85,B 0,C 180,E1 15773.638,E2 15773.638} C_VEL
LIN {X 0,Y 434.667,Z 1132.427,A -85,B 0,C 180,E1 15770.576,E2 15770.576} C_VEL
LIN {X 0,Y 433.522,Z 1142.434,A -85,B 0,C 180,E1 15767.725,E2 15767.725} C_VEL
LIN {X 0,Y 432.744,Z 1150.698,A -85,B 0,C 180,E1 15764.861,E2 15764.861} C_VEL
LIN {X 0,Y 432.278,Z 1157.653,A -85,B 0,C 180,E1 15761.933,E2 15761.933} C_VEL
LIN {X 0,Y 432.035,Z 1163.049,A -85,B 0,C 180,E1 15758.92,E2 15758.92} C_VEL
LIN {X 0,Y 431.924,Z 1166.757,A -85,B 0,C 180,E1 15756.113,E2 15756.113} C_VEL
LIN {X 0,Y 431.886,Z 1169.052,A -85,B 0,C 180,E1 15753.185,E2 15753.185} C_VEL
LIN {X 0,Y 431.885,Z 1169.894,A -85,B 0,C 180,E1 15750.663,E2 15750.663} C_VEL
LIN {X 0,Y 431.911,Z 1169.46,A -85,B 0,C 180,E1 15747.612,E2 15747.612} C_VEL
LIN {X 0,Y 431.918,Z 1167.727,A -85,B 0,C 180,E1 15744.953,E2 15744.953} C_VEL
LIN {X 0,Y 431.996,Z 1164.494,A -85,B 0,C 180,E1 15742.017,E2 15742.017} C_VEL
LIN {X 0,Y 432.177,Z 1159.573,A -85,B 0,C 180,E1 15739.064,E2 15739.064} C_VEL
LIN {X 0,Y 432.557,Z 1153.168,A -85,B 0,C 180,E1 15736.09,E2 15736.09} C_VEL
LIN {X 0,Y 433.212,Z 1145.335,A -85,B 0,C 180,E1 15733.232,E2 15733.232} C_VEL
LIN {X 0,Y 434.291,Z 1135.409,A -85,B 0,C 180,E1 15730.218,E2 15730.218} C_VEL
LIN {X 0,Y 435.622,Z 1125.14,A -85,B 0,C 180,E1 15727.604,E2 15727.604} C_VEL
LIN {X 0,Y 437.262,Z 1113.756,A -85,B 0,C 180,E1 15725.119,E2 15725.119} C_VEL
LIN {X 0,Y 439.306,Z 1099.885,A -85,B 0,C 180,E1 15722.577,E2 15722.577} C_VEL
LIN {X 0,Y 441.863,Z 1083.55,A -85,B 0,C 180,E1 15719.994,E2 15719.994} C_VEL
LIN {X 0,Y 444.463,Z 1067.321,A -85,B 0,C 180,E1 15717.781,E2 15717.781} C_VEL
LIN {X 0,Y 447.258,Z 1049.617,A -85,B 0,C 180,E1 15715.712,E2 15715.712} C_VEL
LIN {X 0,Y 450.172,Z 1030.589,A -85,B 0,C 180,E1 15713.786,E2 15713.786} C_VEL
LIN {X 0,Y 453.072,Z 1010.551,A -85,B 0,C 180,E1 15712.077,E2 15712.077} C_VEL
LIN {X 0,Y 455.982,Z 989.011,A -85,B 0,C 180,E1 15710.513,E2 15710.513} C_VEL
LIN {X 0,Y 458.552,Z 967.773,A -85,B 0,C 180,E1 15709.228,E2 15709.228} C_VEL
LIN {X 0,Y 460.982,Z 945.409,A -85,B 0,C 180,E1 15708.125,E2 15708.125} C_VEL
LIN {X 0,Y 463.122,Z 922.735,A -85,B 0,C 180,E1 15707.229,E2 15707.229} C_VEL
LIN {X 0,Y 464.698,Z 900.725,A -85,B 0,C 180,E1 15706.587,E2 15706.587} C_VEL
LIN {X 0,Y 465.874,Z 875.547,A -85,B 0,C 180,E1 15706.058,E2 15706.058} C_VEL
LIN {X 0,Y 472.478,Z 664.199,A -85,B 0,C 180,E1 15702.246,E2 15702.246} C_VEL
LIN {X 0,Y 474.673,Z 593.294,A -85,B 0,C 180,E1 15700.946,E2 15700.946} C_VEL
LIN {X 0,Y 462.714,Z 575.168,A -85,B 0,C 180,E1 15698.94,E2 15698.94} C_VEL
LIN {X 0,Y 452.926,Z 561.332,A -85,B 0,C 180,E1 15697.179,E2 15697.179} C_VEL
LIN {X 0,Y 444.833,Z 550.408,A -85,B 0,C 180,E1 15695.602,E2 15695.602} C_VEL
LIN {X 0,Y 440.787,Z 543.143,A -85,B 0,C 180,E1 15694.075,E2 15694.075} C_VEL
LIN {X 0,Y 438.212,Z 538.5,A -85,B 0,C 180,E1 15693.046,E2 15693.046} C_VEL
LIN {X 0,Y 435.736,Z 533.963,A -85,B 0,C 180,E1 15692.009,E2 15692.009} C_VEL
LIN {X 0,Y 433.69,Z 530.855,A -85,B 0,C 180,E1 15691.204,E2 15691.204} C_VEL
LIN {X 0,Y 433.29,Z 529.288,A -85,B 0,C 180,E1 15690.816,E2 15690.816} C_VEL
LIN {X 0,Y 433.245,Z 529.033,A -85,B 0,C 180,E1 15687.022,E2 15687.022} C_VEL
LIN {X 0,Y 433.253,Z 529.05,A -85,B 0,C 180,E1 15683.243,E2 15683.243} C_VEL
LIN {X 0,Y 433.248,Z 529.067,A -85,B 0,C 180,E1 15679.41,E2 15679.41} C_VEL
LIN {X 0,Y 433.244,Z 529.024,A -85,B 0,C 180,E1 15675.528,E2 15675.528} C_VEL
LIN {X 0,Y 433.253,Z 529.077,A -85,B 0,C 180,E1 15671.717,E2 15671.717} C_VEL
LIN {X 0,Y 433.242,Z 529.027,A -85,B 0,C 180,E1 15667.826,E2 15667.826} C_VEL
LIN {X 0,Y 433.245,Z 529.069,A -85,B 0,C 180,E1 15663.97,E2 15663.97} C_VEL
LIN {X 0,Y 433.26,Z 529.067,A -85,B 0,C 180,E1 15660.132,E2 15660.132} C_VEL
LIN {X 0,Y 433.249,Z 529.068,A -85,B 0,C 180,E1 15656.295,E2 15656.295} C_VEL
LIN {X 0,Y 433.256,Z 529.064,A -85,B 0,C 180,E1 15652.441,E2 15652.441} C_VEL
LIN {X 0,Y 433.24,Z 529.038,A -85,B 0,C 180,E1 15648.687,E2 15648.687} C_VEL
LIN {X 0,Y 433.242,Z 529.07,A -85,B 0,C 180,E1 15644.883,E2 15644.883} C_VEL
LIN {X 0,Y 433.251,Z 529.026,A -85,B 0,C 180,E1 15641.121,E2 15641.121} C_VEL
LIN {X 0,Y 433.253,Z 529.08,A -85,B 0,C 180,E1 15637.331,E2 15637.331} C_VEL
LIN {X 0,Y 433.251,Z 529.038,A -85,B 0,C 180,E1 15633.55,E2 15633.55} C_VEL
LIN {X 0,Y 433.235,Z 529.04,A -85,B 0,C 180,E1 15629.936,E2 15629.936} C_VEL
LIN {X 0,Y 433.289,Z 529.324,A -85,B 0,C 180,E1 15626.736,E2 15626.736} C_VEL
LIN {X 0,Y 434.801,Z 532.906,A -85,B 0,C 180,E1 15625.868,E2 15625.868} C_VEL
LIN {X 0,Y 436.164,Z 534.761,A -85,B 0,C 180,E1 15625.353,E2 15625.353} C_VEL
LIN {X 0,Y 438.328,Z 538.696,A -85,B 0,C 180,E1 15624.431,E2 15624.431} C_VEL
LIN {X 0,Y 444.113,Z 549.481,A -85,B 0,C 180,E1 15622.075,E2 15622.075} C_VEL
LIN {X 0,Y 450.703,Z 562.311,A -85,B 0,C 180,E1 15619.546,E2 15619.546} C_VEL
LIN {X 0,Y 457.934,Z 577.454,A -85,B 0,C 180,E1 15616.889,E2 15616.889} C_VEL
LIN {X 0,Y 461.293,Z 584.645,A -85,B 0,C 180,E1 15615.781,E2 15615.781} C_VEL
LIN {X 0,Y 465.586,Z 591.725,A -85,B 0,C 180,E1 15615.035,E2 15615.035} C_VEL
LIN {X 0,Y 470.336,Z 623.922,A -85,B 0,C 180,E1 15613.725,E2 15613.725} C_VEL
LIN {X 0,Y 464.73,Z 843.27,A -85,B 0,C 180,E1 15610.029,E2 15610.029} C_VEL
LIN {X 0,Y 463.821,Z 850.974,A -85,B 0,C 180,E1 15609.984,E2 15609.984} C_VEL
LIN {X 0,Y 458.724,Z 871.551,A -85,B 0,C 180,E1 15610.171,E2 15610.171} C_VEL
LIN {X 0,Y 458.021,Z 878.161,A -85,B 0,C 180,E1 15610.123,E2 15610.123} C_VEL
LIN {X 0,Y 456.962,Z 903.911,A -85,B 0,C 180,E1 15609.619,E2 15609.619} C_VEL
LIN {X 0,Y 455.46,Z 924.875,A -85,B 0,C 180,E1 15609.012,E2 15609.012} C_VEL
LIN {X 0,Y 453.444,Z 945.009,A -85,B 0,C 180,E1 15608.208,E2 15608.208} C_VEL
LIN {X 0,Y 450.82,Z 966.511,A -85,B 0,C 180,E1 15607.104,E2 15607.104} C_VEL
LIN {X 0,Y 448.09,Z 986.031,A -85,B 0,C 180,E1 15605.855,E2 15605.855} C_VEL
LIN {X 0,Y 445.049,Z 1004.56,A -85,B 0,C 180,E1 15604.404,E2 15604.404} C_VEL
LIN {X 0,Y 441.665,Z 1023.75,A -85,B 0,C 180,E1 15602.602,E2 15602.602} C_VEL
LIN {X 0,Y 438.553,Z 1040.453,A -85,B 0,C 180,E1 15600.737,E2 15600.737} C_VEL
LIN {X 0,Y 435.402,Z 1056.432,A -85,B 0,C 180,E1 15598.607,E2 15598.607} C_VEL
LIN {X 0,Y 432.453,Z 1071.784,A -85,B 0,C 180,E1 15596.206,E2 15596.206} C_VEL
LIN {X 0,Y 429.991,Z 1085.358,A -85,B 0,C 180,E1 15593.721,E2 15593.721} C_VEL
LIN {X 0,Y 427.948,Z 1097.555,A -85,B 0,C 180,E1 15591.088,E2 15591.088} C_VEL
LIN {X 0,Y 426.359,Z 1108.378,A -85,B 0,C 180,E1 15588.315,E2 15588.315} C_VEL
LIN {X 0,Y 425.228,Z 1117.834,A -85,B 0,C 180,E1 15585.409,E2 15585.409} C_VEL
LIN {X 0,Y 424.518,Z 1125.495,A -85,B 0,C 180,E1 15582.514,E2 15582.514} C_VEL
LIN {X 0,Y 424.132,Z 1131.39,A -85,B 0,C 180,E1 15579.635,E2 15579.635} C_VEL
LIN {X 0,Y 423.973,Z 1135.918,A -85,B 0,C 180,E1 15576.636,E2 15576.636} C_VEL
LIN {X 0,Y 423.909,Z 1138.682,A -85,B 0,C 180,E1 15573.787,E2 15573.787} C_VEL
LIN {X 0,Y 423.905,Z 1139.895,A -85,B 0,C 180,E1 15570.946,E2 15570.946} C_VEL
LIN {X 0,Y 423.903,Z 1139.74,A -85,B 0,C 180,E1 15568.108,E2 15568.108} C_VEL
LIN {X 0,Y 423.916,Z 1137.98,A -85,B 0,C 180,E1 15565.265,E2 15565.265} C_VEL
LIN {X 0,Y 423.992,Z 1134.593,A -85,B 0,C 180,E1 15562.275,E2 15562.275} C_VEL
LIN {X 0,Y 424.21,Z 1130.067,A -85,B 0,C 180,E1 15559.543,E2 15559.543} C_VEL
LIN {X 0,Y 424.67,Z 1123.661,A -85,B 0,C 180,E1 15556.66,E2 15556.66} C_VEL
LIN {X 0,Y 425.478,Z 1115.606,A -85,B 0,C 180,E1 15553.761,E2 15553.761} C_VEL
LIN {X 0,Y 426.743,Z 1105.713,A -85,B 0,C 180,E1 15550.851,E2 15550.851} C_VEL
LIN {X 0,Y 428.464,Z 1094.273,A -85,B 0,C 180,E1 15548.076,E2 15548.076} C_VEL
LIN {X 0,Y 430.652,Z 1081.479,A -85,B 0,C 180,E1 15545.443,E2 15545.443} C_VEL
LIN {X 0,Y 433.321,Z 1067.333,A -85,B 0,C 180,E1 15542.958,E2 15542.958} C_VEL
LIN {X 0,Y 436.242,Z 1052.18,A -85,B 0,C 180,E1 15540.703,E2 15540.703} C_VEL
LIN {X 0,Y 439.453,Z 1035.555,A -85,B 0,C 180,E1 15538.599,E2 15538.599} C_VEL
LIN {X 0,Y 442.631,Z 1018.617,A -85,B 0,C 180,E1 15536.785,E2 15536.785} C_VEL
LIN {X 0,Y 445.675,Z 1000.891,A -85,B 0,C 180,E1 15535.197,E2 15535.197} C_VEL
LIN {X 0,Y 448.756,Z 981.249,A -85,B 0,C 180,E1 15533.729,E2 15533.729} C_VEL
LIN {X 0,Y 451.434,Z 962.224,A -85,B 0,C 180,E1 15532.556,E2 15532.556} C_VEL
LIN {X 0,Y 453.754,Z 942.281,A -85,B 0,C 180,E1 15531.582,E2 15531.582} C_VEL
LIN {X 0,Y 455.779,Z 920.762,A -85,B 0,C 180,E1 15530.763,E2 15530.763} C_VEL
LIN {X 0,Y 457.19,Z 900.458,A -85,B 0,C 180,E1 15530.206,E2 15530.206} C_VEL
LIN {X 0,Y 458.287,Z 867.534,A -85,B 0,C 180,E1 15529.606,E2 15529.606} C_VEL
LIN {X 0,Y 464.294,Z 642.497,A -85,B 0,C 180,E1 15525.787,E2 15525.787} C_VEL
LIN {X 0,Y 464.515,Z 628.844,A -85,B 0,C 180,E1 15525.524,E2 15525.524} C_VEL
LIN {X 0,Y 458.195,Z 595.865,A -85,B 0,C 180,E1 15523.936,E2 15523.936} C_VEL
LIN {X 0,Y 450.4,Z 583.28,A -85,B 0,C 180,E1 15522.444,E2 15522.444} C_VEL
LIN {X 0,Y 444.228,Z 568.895,A -85,B 0,C 180,E1 15519.659,E2 15519.659} C_VEL
LIN {X 0,Y 439.97,Z 568.576,A -85,B 0,C 180,E1 15518.846,E2 15518.846} C_VEL
LIN {X 0,Y 440.002,Z 569.458,A -85,B 0,C 180,E1 15518.637,E2 15518.637} C_VEL
LIN {X 0,Y 441.287,Z 573.826,A -85,B 0,C 180,E1 15518.129,E2 15518.129} C_VEL
LIN {X 0,Y 439.448,Z 616.856,A -85,B 0,C 180,E1 15514.431,E2 15514.431} C_VEL
LIN {X 0,Y 437.662,Z 657.622,A -85,B 0,C 180,E1 15510.933,E2 15510.933} C_VEL
LIN {X 0,Y 435.63,Z 700.618,A -85,B 0,C 180,E1 15507.252,E2 15507.252} C_VEL
LIN {X 0,Y 434.946,Z 719.324,A -85,B 0,C 180,E1 15505.701,E2 15505.701} C_VEL
LIN {X 0,Y 435.774,Z 728.469,A -85,B 0,C 180,E1 15505.467,E2 15505.467} C_VEL
LIN {X 0,Y 432.739,Z 890.964,A -85,B 0,C 180,E1 15502.457,E2 15502.457} C_VEL
LIN {X 0,Y 432.32,Z 908.584,A -85,B 0,C 180,E1 15501.879,E2 15501.879} C_VEL
LIN {X 0,Y 431.636,Z 926.156,A -85,B 0,C 180,E1 15501.042,E2 15501.042} C_VEL
LIN {X 0,Y 430.837,Z 942.282,A -85,B 0,C 180,E1 15500.018,E2 15500.018} C_VEL
LIN {X 0,Y 429.925,Z 957.028,A -85,B 0,C 180,E1 15498.818,E2 15498.818} C_VEL
LIN {X 0,Y 428.946,Z 971.416,A -85,B 0,C 180,E1 15497.36,E2 15497.36} C_VEL
LIN {X 0,Y 427.99,Z 984.547,A -85,B 0,C 180,E1 15495.724,E2 15495.724} C_VEL
LIN {X 0,Y 427.12,Z 996.049,A -85,B 0,C 180,E1 15493.953,E2 15493.953} C_VEL
LIN {X 0,Y 426.391,Z 1006.068,A -85,B 0,C 180,E1 15492.046,E2 15492.046} C_VEL
LIN {X 0,Y 425.821,Z 1014.67,A -85,B 0,C 180,E1 15490.007,E2 15490.007} C_VEL
LIN {X 0,Y 425.411,Z 1021.792,A -85,B 0,C 180,E1 15487.835,E2 15487.835} C_VEL
LIN {X 0,Y 425.159,Z 1027.266,A -85,B 0,C 180,E1 15485.533,E2 15485.533} C_VEL
LIN {X 0,Y 425.059,Z 1030.918,A -85,B 0,C 180,E1 15483.237,E2 15483.237} C_VEL
LIN {X 0,Y 425.059,Z 1032.832,A -85,B 0,C 180,E1 15480.944,E2 15480.944} C_VEL
LIN {X 0,Y 425.114,Z 1032.989,A -85,B 0,C 180,E1 15478.653,E2 15478.653} C_VEL
LIN {X 0,Y 425.231,Z 1031.46,A -85,B 0,C 180,E1 15476.36,E2 15476.36} C_VEL
LIN {X 0,Y 425.463,Z 1028.188,A -85,B 0,C 180,E1 15474.065,E2 15474.065} C_VEL
LIN {X 0,Y 425.806,Z 1023.31,A -85,B 0,C 180,E1 15471.901,E2 15471.901} C_VEL
LIN {X 0,Y 426.329,Z 1016.535,A -85,B 0,C 180,E1 15469.733,E2 15469.733} C_VEL
LIN {X 0,Y 426.986,Z 1008.22,A -85,B 0,C 180,E1 15467.697,E2 15467.697} C_VEL
LIN {X 0,Y 427.706,Z 999.095,A -85,B 0,C 180,E1 15465.929,E2 15465.929} C_VEL
LIN {X 0,Y 428.572,Z 987.687,A -85,B 0,C 180,E1 15464.16,E2 15464.16} C_VEL
LIN {X 0,Y 429.468,Z 975.186,A -85,B 0,C 180,E1 15462.593,E2 15462.593} C_VEL
LIN {X 0,Y 430.302,Z 961.668,A -85,B 0,C 180,E1 15461.227,E2 15461.227} C_VEL
LIN {X 0,Y 431.012,Z 947.096,A -85,B 0,C 180,E1 15460.062,E2 15460.062} C_VEL
LIN {X 0,Y 431.66,Z 930.472,A -85,B 0,C 180,E1 15459.031,E2 15459.031} C_VEL
LIN {X 0,Y 432.085,Z 913.726,A -85,B 0,C 180,E1 15458.27,E2 15458.27} C_VEL
LIN {X 0,Y 432.271,Z 895.663,A -85,B 0,C 180,E1 15457.726,E2 15457.726} C_VEL
LIN {X 0,Y 434.073,Z 790.59,A -85,B 0,C 180,E1 15455.723,E2 15455.723} C_VEL
LIN {X 0,Y 435.749,Z 732.66,A -85,B 0,C 180,E1 15454.518,E2 15454.518} C_VEL
LIN {X 0,Y 436.883,Z 726.186,A -85,B 0,C 180,E1 15454.08,E2 15454.08} C_VEL
LIN {X 0,Y 438.129,Z 684.586,A -85,B 0,C 180,E1 15450.767,E2 15450.767} C_VEL
LIN {X 0,Y 438.992,Z 643.969,A -85,B 0,C 180,E1 15447.64,E2 15447.64} C_VEL
LIN {X 0,Y 439.62,Z 597.672,A -85,B 0,C 180,E1 15444.192,E2 15444.192} C_VEL
LIN {X 0,Y 440.503,Z 595.868,A -85,B 0,C 180,E1 15443.913,E2 15443.913} C_VEL
LIN {X 0,Y 443.335,Z 593.7,A -85,B 0,C 180,E1 15443.499,E2 15443.499} C_VEL
LIN {X 0,Y 446.673,Z 588.874,A -85,B 0,C 180,E1 15443.097,E2 15443.097} C_VEL
LIN {X 0,Y 448.808,Z 585.1,A -85,B 0,C 180,E1 15442.863,E2 15442.863} C_VEL
LIN {X 0,Y 452.574,Z 581.97,A -85,B 0,C 180,E1 15442.369,E2 15442.369} C_VEL
LIN {X 0,Y 455.639,Z 578.045,A -85,B 0,C 180,E1 15442.01,E2 15442.01} C_VEL
LIN {X 0,Y 468.666,Z 597.874,A -85,B 0,C 180,E1 15439.728,E2 15439.728} C_VEL
LIN {X 0,Y 469.059,Z 599.09,A -85,B 0,C 180,E1 15439.649,E2 15439.649} C_VEL
LIN {X 0,Y 461.894,Z 811.737,A -85,B 0,C 180,E1 15435.757,E2 15435.757} C_VEL
LIN {X 0,Y 459.098,Z 893.143,A -85,B 0,C 180,E1 15434.25,E2 15434.25} C_VEL
LIN {X 0,Y 457.432,Z 916.172,A -85,B 0,C 180,E1 15433.624,E2 15433.624} C_VEL
LIN {X 0,Y 455.336,Z 939.348,A -85,B 0,C 180,E1 15432.772,E2 15432.772} C_VEL
LIN {X 0,Y 453.039,Z 959.92,A -85,B 0,C 180,E1 15431.799,E2 15431.799} C_VEL
LIN {X 0,Y 450.194,Z 982.184,A -85,B 0,C 180,E1 15430.514,E2 15430.514} C_VEL
LIN {X 0,Y 447.182,Z 1003.83,A -85,B 0,C 180,E1 15429.007,E2 15429.007} C_VEL
LIN {X 0,Y 444.181,Z 1023.838,A -85,B 0,C 180,E1 15427.348,E2 15427.348} C_VEL
LIN {X 0,Y 441.256,Z 1042.46,A -85,B 0,C 180,E1 15425.564,E2 15425.564} C_VEL
LIN {X 0,Y 438.233,Z 1060.635,A -85,B 0,C 180,E1 15423.514,E2 15423.514} C_VEL
LIN {X 0,Y 435.27,Z 1078.505,A -85,B 0,C 180,E1 15421.184,E2 15421.184} C_VEL
LIN {X 0,Y 432.871,Z 1092.781,A -85,B 0,C 180,E1 15419.017,E2 15419.017} C_VEL
LIN {X 0,Y 430.345,Z 1108.477,A -85,B 0,C 180,E1 15416.257,E2 15416.257} C_VEL
LIN {X 0,Y 428.456,Z 1121.147,A -85,B 0,C 180,E1 15413.665,E2 15413.665} C_VEL
LIN {X 0,Y 426.846,Z 1132.893,A -85,B 0,C 180,E1 15410.833,E2 15410.833} C_VEL
LIN {X 0,Y 425.675,Z 1142.433,A -85,B 0,C 180,E1 15408.062,E2 15408.062} C_VEL
LIN {X 0,Y 424.83,Z 1150.697,A -85,B 0,C 180,E1 15405.144,E2 15405.144} C_VEL
LIN {X 0,Y 424.323,Z 1157.468,A -85,B 0,C 180,E1 15402.244,E2 15402.244} C_VEL
LIN {X 0,Y 424.053,Z 1162.842,A -85,B 0,C 180,E1 15399.226,E2 15399.226} C_VEL
LIN {X 0,Y 423.945,Z 1166.438,A -85,B 0,C 180,E1 15396.5,E2 15396.5} C_VEL
LIN {X 0,Y 423.888,Z 1168.984,A -85,B 0,C 180,E1 15393.381,E2 15393.381} C_VEL
LIN {X 0,Y 423.887,Z 1169.871,A -85,B 0,C 180,E1 15390.811,E2 15390.811} C_VEL
LIN {X 0,Y 423.911,Z 1169.595,A -85,B 0,C 180,E1 15387.837,E2 15387.837} C_VEL
LIN {X 0,Y 423.917,Z 1167.84,A -85,B 0,C 180,E1 15384.993,E2 15384.993} C_VEL
LIN {X 0,Y 423.999,Z 1164.68,A -85,B 0,C 180,E1 15382.002,E2 15382.002} C_VEL
LIN {X 0,Y 424.191,Z 1159.827,A -85,B 0,C 180,E1 15378.993,E2 15378.993} C_VEL
LIN {X 0,Y 424.596,Z 1153.516,A -85,B 0,C 180,E1 15375.963,E2 15375.963} C_VEL
LIN {X 0,Y 425.295,Z 1145.739,A -85,B 0,C 180,E1 15373.051,E2 15373.051} C_VEL
LIN {X 0,Y 426.396,Z 1136.362,A -85,B 0,C 180,E1 15370.102,E2 15370.102} C_VEL
LIN {X 0,Y 427.669,Z 1126.615,A -85,B 0,C 180,E1 15367.599,E2 15367.599} C_VEL
LIN {X 0,Y 429.442,Z 1114.505,A -85,B 0,C 180,E1 15364.916,E2 15364.916} C_VEL
LIN {X 0,Y 431.671,Z 1100.169,A -85,B 0,C 180,E1 15362.227,E2 15362.227} C_VEL
LIN {X 0,Y 434.251,Z 1084.617,A -85,B 0,C 180,E1 15359.703,E2 15359.703} C_VEL
LIN {X 0,Y 436.836,Z 1069.057,A -85,B 0,C 180,E1 15357.538,E2 15357.538} C_VEL
LIN {X 0,Y 440.045,Z 1049.752,A -85,B 0,C 180,E1 15355.228,E2 15355.228} C_VEL
LIN {X 0,Y 443.11,Z 1030.76,A -85,B 0,C 180,E1 15353.276,E2 15353.276} C_VEL
LIN {X 0,Y 446.156,Z 1010.795,A -85,B 0,C 180,E1 15351.545,E2 15351.545} C_VEL
LIN {X 0,Y 449.217,Z 989.479,A -85,B 0,C 180,E1 15349.965,E2 15349.965} C_VEL
LIN {X 0,Y 451.943,Z 968.649,A -85,B 0,C 180,E1 15348.67,E2 15348.67} C_VEL
LIN {X 0,Y 454.597,Z 946.12,A -85,B 0,C 180,E1 15347.528,E2 15347.528} C_VEL
LIN {X 0,Y 456.759,Z 924.554,A -85,B 0,C 180,E1 15346.654,E2 15346.654} C_VEL
LIN {X 0,Y 458.518,Z 902.013,A -85,B 0,C 180,E1 15345.972,E2 15345.972} C_VEL
LIN {X 0,Y 459.756,Z 878.43,A -85,B 0,C 180,E1 15345.455,E2 15345.455} C_VEL
LIN {X 0,Y 466.774,Z 666.51,A -85,B 0,C 180,E1 15341.59,E2 15341.59} C_VEL
LIN {X 0,Y 469.014,Z 596.891,A -85,B 0,C 180,E1 15340.296,E2 15340.296} C_VEL
LIN {X 0,Y 456.594,Z 578.026,A -85,B 0,C 180,E1 15338.135,E2 15338.135} C_VEL
LIN {X 0,Y 444.835,Z 561.639,A -85,B 0,C 180,E1 15335.919,E2 15335.919} C_VEL
LIN {X 0,Y 436.877,Z 551.006,A -85,B 0,C 180,E1 15334.263,E2 15334.263} C_VEL
LIN {X 0,Y 433.304,Z 544.625,A -85,B 0,C 180,E1 15332.838,E2 15332.838} C_VEL
LIN {X 0,Y 430.483,Z 539.699,A -85,B 0,C 180,E1 15331.662,E2 15331.662} C_VEL
LIN {X 0,Y 428.406,Z 535.895,A -85,B 0,C 180,E1 15330.738,E2 15330.738} C_VEL
LIN {X 0,Y 425.883,Z 532.183,A -85,B 0,C 180,E1 15329.694,E2 15329.694} C_VEL
LIN {X 0,Y 425.34,Z 530.274,A -85,B 0,C 180,E1 15329.186,E2 15329.186} C_VEL
LIN {X 0,Y 425.308,Z 530.041,A -85,B 0,C 180,E1 15325.63,E2 15325.63} C_VEL
LIN {X 0,Y 425.305,Z 530.015,A -85,B 0,C 180,E1 15321.779,E2 15321.779} C_VEL
LIN {X 0,Y 425.315,Z 530.061,A -85,B 0,C 180,E1 15317.936,E2 15317.936} C_VEL
LIN {X 0,Y 425.302,Z 530.021,A -85,B 0,C 180,E1 15314.152,E2 15314.152} C_VEL
LIN {X 0,Y 425.305,Z 530.03,A -85,B 0,C 180,E1 15310.292,E2 15310.292} C_VEL
LIN {X 0,Y 425.315,Z 530.043,A -85,B 0,C 180,E1 15306.479,E2 15306.479} C_VEL
LIN {X 0,Y 425.309,Z 530.058,A -85,B 0,C 180,E1 15302.56,E2 15302.56} C_VEL
LIN {X 0,Y 425.314,Z 530.064,A -85,B 0,C 180,E1 15298.653,E2 15298.653} C_VEL
LIN {X 0,Y 425.316,Z 530.068,A -85,B 0,C 180,E1 15294.739,E2 15294.739} C_VEL
LIN {X 0,Y 425.306,Z 530.07,A -85,B 0,C 180,E1 15290.891,E2 15290.891} C_VEL
LIN {X 0,Y 425.298,Z 530.012,A -85,B 0,C 180,E1 15286.956,E2 15286.956} C_VEL
LIN {X 0,Y 425.313,Z 530.059,A -85,B 0,C 180,E1 15283.192,E2 15283.192} C_VEL
LIN {X 0,Y 425.311,Z 530.027,A -85,B 0,C 180,E1 15279.335,E2 15279.335} C_VEL
LIN {X 0,Y 425.311,Z 530.023,A -85,B 0,C 180,E1 15275.559,E2 15275.559} C_VEL
LIN {X 0,Y 425.313,Z 530.071,A -85,B 0,C 180,E1 15271.648,E2 15271.648} C_VEL
LIN {X 0,Y 425.348,Z 530.292,A -85,B 0,C 180,E1 15268.357,E2 15268.357} C_VEL
LIN {X 0,Y 426.891,Z 533.914,A -85,B 0,C 180,E1 15267.404,E2 15267.404} C_VEL
LIN {X 0,Y 428.232,Z 535.582,A -85,B 0,C 180,E1 15266.882,E2 15266.882} C_VEL
LIN {X 0,Y 430.225,Z 539.483,A -85,B 0,C 180,E1 15265.937,E2 15265.937} C_VEL
LIN {X 0,Y 431.453,Z 541.628,A -85,B 0,C 180,E1 15265.405,E2 15265.405} C_VEL
LIN {X 0,Y 434.233,Z 546.717,A -85,B 0,C 180,E1 15264.207,E2 15264.207} C_VEL
LIN {X 0,Y 438.764,Z 555.016,A -85,B 0,C 180,E1 15262.358,E2 15262.358} C_VEL
LIN {X 0,Y 445.344,Z 568.041,A -85,B 0,C 180,E1 15259.76,E2 15259.76} C_VEL
LIN {X 0,Y 452.518,Z 583.168,A -85,B 0,C 180,E1 15257.092,E2 15257.092} C_VEL
LIN {X 0,Y 460.607,Z 596.289,A -85,B 0,C 180,E1 15255.619,E2 15255.619} C_VEL
LIN {X 0,Y 464.78,Z 625.641,A -85,B 0,C 180,E1 15254.412,E2 15254.412} C_VEL
LIN {X 0,Y 458.514,Z 857.908,A -85,B 0,C 180,E1 15250.464,E2 15250.464} C_VEL
LIN {X 0,Y 458.021,Z 878.161,A -85,B 0,C 180,E1 15250.123,E2 15250.123} C_VEL
LIN {X 0,Y 457.097,Z 885.866,A -85,B 0,C 180,E1 15250.077,E2 15250.077} C_VEL
LIN {X 0,Y 451.794,Z 905.262,A -85,B 0,C 180,E1 15250.196,E2 15250.196} C_VEL
LIN {X 0,Y 450.46,Z 912.84,A -85,B 0,C 180,E1 15250.077,E2 15250.077} C_VEL
LIN {X 0,Y 448.579,Z 933.938,A -85,B 0,C 180,E1 15249.361,E2 15249.361} C_VEL
LIN {X 0,Y 446.286,Z 954.306,A -85,B 0,C 180,E1 15248.441,E2 15248.441} C_VEL
LIN {X 0,Y 443.611,Z 974.157,A -85,B 0,C 180,E1 15247.323,E2 15247.323} C_VEL
LIN {X 0,Y 440.583,Z 993.057,A -85,B 0,C 180,E1 15245.999,E2 15245.999} C_VEL
LIN {X 0,Y 437.16,Z 1012.655,A -85,B 0,C 180,E1 15244.343,E2 15244.343} C_VEL
LIN {X 0,Y 433.817,Z 1030.447,A -85,B 0,C 180,E1 15242.548,E2 15242.548} C_VEL
LIN {X 0,Y 430.501,Z 1046.818,A -85,B 0,C 180,E1 15240.573,E2 15240.573} C_VEL
LIN {X 0,Y 427.306,Z 1062.412,A -85,B 0,C 180,E1 15238.36,E2 15238.36} C_VEL
LIN {X 0,Y 424.428,Z 1076.62,A -85,B 0,C 180,E1 15235.988,E2 15235.988} C_VEL
LIN {X 0,Y 421.798,Z 1090.078,A -85,B 0,C 180,E1 15233.32,E2 15233.32} C_VEL
LIN {X 0,Y 419.683,Z 1102.101,A -85,B 0,C 180,E1 15230.501,E2 15230.501} C_VEL
LIN {X 0,Y 418.16,Z 1112.273,A -85,B 0,C 180,E1 15227.678,E2 15227.678} C_VEL
LIN {X 0,Y 417.08,Z 1121.009,A -85,B 0,C 180,E1 15224.721,E2 15224.721} C_VEL
LIN {X 0,Y 416.435,Z 1127.975,A -85,B 0,C 180,E1 15221.776,E2 15221.776} C_VEL
LIN {X 0,Y 416.105,Z 1133.388,A -85,B 0,C 180,E1 15218.846,E2 15218.846} C_VEL
LIN {X 0,Y 415.956,Z 1137.164,A -85,B 0,C 180,E1 15215.933,E2 15215.933} C_VEL
LIN {X 0,Y 415.904,Z 1139.526,A -85,B 0,C 180,E1 15212.894,E2 15212.894} C_VEL
LIN {X 0,Y 415.918,Z 1140.343,A -85,B 0,C 180,E1 15210,E2 15210} C_VEL
LIN {X 0,Y 415.903,Z 1139.569,A -85,B 0,C 180,E1 15207.106,E2 15207.106} C_VEL
LIN {X 0,Y 415.951,Z 1137.419,A -85,B 0,C 180,E1 15204.206,E2 15204.206} C_VEL
LIN {X 0,Y 416.078,Z 1133.916,A -85,B 0,C 180,E1 15201.432,E2 15201.432} C_VEL
LIN {X 0,Y 416.401,Z 1128.454,A -85,B 0,C 180,E1 15198.364,E2 15198.364} C_VEL
LIN {X 0,Y 417.025,Z 1121.646,A -85,B 0,C 180,E1 15195.419,E2 15195.419} C_VEL
LIN {X 0,Y 418.051,Z 1112.983,A -85,B 0,C 180,E1 15192.461,E2 15192.461} C_VEL
LIN {X 0,Y 419.536,Z 1102.986,A -85,B 0,C 180,E1 15189.638,E2 15189.638} C_VEL
LIN {X 0,Y 421.5,Z 1091.815,A -85,B 0,C 180,E1 15186.958,E2 15186.958} C_VEL
LIN {X 0,Y 424.028,Z 1078.555,A -85,B 0,C 180,E1 15184.286,E2 15184.286} C_VEL
LIN {X 0,Y 426.825,Z 1064.703,A -85,B 0,C 180,E1 15181.91,E2 15181.91} C_VEL
LIN {X 0,Y 429.874,Z 1050.113,A -85,B 0,C 180,E1 15179.764,E2 15179.764} C_VEL
LIN {X 0,Y 433.071,Z 1034.007,A -85,B 0,C 180,E1 15177.769,E2 15177.769} C_VEL
LIN {X 0,Y 436.581,Z 1015.852,A -85,B 0,C 180,E1 15175.868,E2 15175.868} C_VEL
LIN {X 0,Y 439.863,Z 997.575,A -85,B 0,C 180,E1 15174.254,E2 15174.254} C_VEL
LIN {X 0,Y 442.96,Z 978.248,A -85,B 0,C 180,E1 15172.857,E2 15172.857} C_VEL
LIN {X 0,Y 445.793,Z 958.273,A -85,B 0,C 180,E1 15171.672,E2 15171.672} C_VEL
LIN {X 0,Y 448.091,Z 939.068,A -85,B 0,C 180,E1 15170.758,E2 15170.758} C_VEL
LIN {X 0,Y 450.065,Z 917.638,A -85,B 0,C 180,E1 15169.978,E2 15169.978} C_VEL
LIN {X 0,Y 451.558,Z 895.864,A -85,B 0,C 180,E1 15169.417,E2 15169.417} C_VEL
LIN {X 0,Y 457.494,Z 685.948,A -85,B 0,C 180,E1 15165.81,E2 15165.81} C_VEL
LIN {X 0,Y 459.06,Z 630.8,A -85,B 0,C 180,E1 15164.831,E2 15164.831} C_VEL
LIN {X 0,Y 453.379,Z 600.589,A -85,B 0,C 180,E1 15163.347,E2 15163.347} C_VEL
LIN {X 0,Y 442.254,Z 582.926,A -85,B 0,C 180,E1 15161.183,E2 15161.183} C_VEL
LIN {X 0,Y 438.893,Z 575.435,A -85,B 0,C 180,E1 15159.677,E2 15159.677} C_VEL
LIN {X 0,Y 434.117,Z 575.096,A -85,B 0,C 180,E1 15158.791,E2 15158.791} C_VEL
LIN {X 0,Y 434.059,Z 575.91,A -85,B 0,C 180,E1 15158.562,E2 15158.562} C_VEL
LIN {X 0,Y 433.021,Z 602.338,A -85,B 0,C 180,E1 15156.236,E2 15156.236} C_VEL
LIN {X 0,Y 431.145,Z 643.779,A -85,B 0,C 180,E1 15152.666,E2 15152.666} C_VEL
LIN {X 0,Y 429.131,Z 686.468,A -85,B 0,C 180,E1 15148.989,E2 15148.989} C_VEL
LIN {X 0,Y 427.613,Z 720.197,A -85,B 0,C 180,E1 15146.118,E2 15146.118} C_VEL
LIN {X 0,Y 428.433,Z 729.257,A -85,B 0,C 180,E1 15145.881,E2 15145.881} C_VEL
LIN {X 0,Y 425.186,Z 892.123,A -85,B 0,C 180,E1 15142.791,E2 15142.791} C_VEL
LIN {X 0,Y 424.75,Z 909.815,A -85,B 0,C 180,E1 15142.199,E2 15142.199} C_VEL
LIN {X 0,Y 424.047,Z 927.325,A -85,B 0,C 180,E1 15141.35,E2 15141.35} C_VEL
LIN {X 0,Y 423.201,Z 943.747,A -85,B 0,C 180,E1 15140.288,E2 15140.288} C_VEL
LIN {X 0,Y 422.21,Z 959.132,A -85,B 0,C 180,E1 15139.004,E2 15139.004} C_VEL
LIN {X 0,Y 421.175,Z 973.793,A -85,B 0,C 180,E1 15137.476,E2 15137.476} C_VEL
LIN {X 0,Y 420.224,Z 986.262,A -85,B 0,C 180,E1 15135.88,E2 15135.88} C_VEL
LIN {X 0,Y 419.317,Z 997.696,A -85,B 0,C 180,E1 15134.077,E2 15134.077} C_VEL
LIN {X 0,Y 418.52,Z 1008.352,A -85,B 0,C 180,E1 15131.997,E2 15131.997} C_VEL
LIN {X 0,Y 417.941,Z 1016.817,A -85,B 0,C 180,E1 15129.919,E2 15129.919} C_VEL
LIN {X 0,Y 417.517,Z 1023.72,A -85,B 0,C 180,E1 15127.707,E2 15127.707} C_VEL
LIN {X 0,Y 417.277,Z 1029.096,A -85,B 0,C 180,E1 15125.362,E2 15125.362} C_VEL
LIN {X 0,Y 417.187,Z 1032.625,A -85,B 0,C 180,E1 15123.023,E2 15123.023} C_VEL
LIN {X 0,Y 417.189,Z 1034.338,A -85,B 0,C 180,E1 15120.687,E2 15120.687} C_VEL
LIN {X 0,Y 417.255,Z 1034.365,A -85,B 0,C 180,E1 15118.353,E2 15118.353} C_VEL
LIN {X 0,Y 417.411,Z 1032.688,A -85,B 0,C 180,E1 15116.017,E2 15116.017} C_VEL
LIN {X 0,Y 417.663,Z 1029.441,A -85,B 0,C 180,E1 15113.816,E2 15113.816} C_VEL
LIN {X 0,Y 418.051,Z 1024.444,A -85,B 0,C 180,E1 15111.611,E2 15111.611} C_VEL
LIN {X 0,Y 418.632,Z 1017.532,A -85,B 0,C 180,E1 15109.403,E2 15109.403} C_VEL
LIN {X 0,Y 419.348,Z 1009.032,A -85,B 0,C 180,E1 15107.329,E2 15107.329} C_VEL
LIN {X 0,Y 420.193,Z 998.869,A -85,B 0,C 180,E1 15105.391,E2 15105.391} C_VEL
LIN {X 0,Y 421.106,Z 987.528,A -85,B 0,C 180,E1 15103.659,E2 15103.659} C_VEL
LIN {X 0,Y 422.013,Z 975.175,A -85,B 0,C 180,E1 15102.133,E2 15102.133} C_VEL
LIN {X 0,Y 422.876,Z 961.115,A -85,B 0,C 180,E1 15100.742,E2 15100.742} C_VEL
LIN {X 0,Y 423.64,Z 945.929,A -85,B 0,C 180,E1 15099.552,E2 15099.552} C_VEL
LIN {X 0,Y 424.244,Z 929.796,A -85,B 0,C 180,E1 15098.582,E2 15098.582} C_VEL
LIN {X 0,Y 424.652,Z 911.987,A -85,B 0,C 180,E1 15097.81,E2 15097.81} C_VEL
LIN {X 0,Y 424.802,Z 894.278,A -85,B 0,C 180,E1 15097.307,E2 15097.307} C_VEL
LIN {X 0,Y 426.512,Z 802.574,A -85,B 0,C 180,E1 15095.513,E2 15095.513} C_VEL
LIN {X 0,Y 428.634,Z 735.057,A -85,B 0,C 180,E1 15094.064,E2 15094.064} C_VEL
LIN {X 0,Y 429.954,Z 728.309,A -85,B 0,C 180,E1 15093.63,E2 15093.63} C_VEL
LIN {X 0,Y 431.334,Z 686.363,A -85,B 0,C 180,E1 15090.26,E2 15090.26} C_VEL
LIN {X 0,Y 432.341,Z 645.456,A -85,B 0,C 180,E1 15087.08,E2 15087.08} C_VEL
LIN {X 0,Y 433.02,Z 615.54,A -85,B 0,C 180,E1 15084.783,E2 15084.783} C_VEL
LIN {X 0,Y 433.982,Z 613.862,A -85,B 0,C 180,E1 15084.509,E2 15084.509} C_VEL
LIN {X 0,Y 436.821,Z 611.429,A -85,B 0,C 180,E1 15084.089,E2 15084.089} C_VEL
LIN {X 0,Y 440.525,Z 605.817,A -85,B 0,C 180,E1 15083.633,E2 15083.633} C_VEL
LIN {X 0,Y 442.238,Z 602.911,A -85,B 0,C 180,E1 15083.435,E2 15083.435} C_VEL
LIN {X 0,Y 445.872,Z 599.92,A -85,B 0,C 180,E1 15082.94,E2 15082.94} C_VEL
LIN {X 0,Y 449.779,Z 594.542,A -85,B 0,C 180,E1 15082.476,E2 15082.476} C_VEL
LIN {X 0,Y 451.713,Z 591.355,A -85,B 0,C 180,E1 15082.264,E2 15082.264} C_VEL
LIN {X 0,Y 454.812,Z 588.777,A -85,B 0,C 180,E1 15081.869,E2 15081.869} C_VEL
LIN {X 0,Y 463.508,Z 602.425,A -85,B 0,C 180,E1 15080.314,E2 15080.314} C_VEL
LIN {X 0,Y 456.008,Z 813.495,A -85,B 0,C 180,E1 15076.413,E2 15076.413} C_VEL
LIN {X 0,Y 453.119,Z 893.059,A -85,B 0,C 180,E1 15074.923,E2 15074.923} C_VEL
LIN {X 0,Y 451.354,Z 916.261,A -85,B 0,C 180,E1 15074.288,E2 15074.288} C_VEL
LIN {X 0,Y 449.134,Z 939.544,A -85,B 0,C 180,E1 15073.42,E2 15073.42} C_VEL
LIN {X 0,Y 446.725,Z 960.009,A -85,B 0,C 180,E1 15072.44,E2 15072.44} C_VEL
LIN {X 0,Y 443.733,Z 982.132,A -85,B 0,C 180,E1 15071.145,E2 15071.145} C_VEL
LIN {X 0,Y 440.666,Z 1002.611,A -85,B 0,C 180,E1 15069.696,E2 15069.696} C_VEL
LIN {X 0,Y 437.333,Z 1023.309,A -85,B 0,C 180,E1 15067.953,E2 15067.953} C_VEL
LIN {X 0,Y 434.111,Z 1042.753,A -85,B 0,C 180,E1 15066.058,E2 15066.058} C_VEL
LIN {X 0,Y 430.958,Z 1060.74,A -85,B 0,C 180,E1 15063.997,E2 15063.997} C_VEL
LIN {X 0,Y 427.777,Z 1078.96,A -85,B 0,C 180,E1 15061.572,E2 15061.572} C_VEL
LIN {X 0,Y 425.159,Z 1093.992,A -85,B 0,C 180,E1 15059.252,E2 15059.252} C_VEL
LIN {X 0,Y 422.657,Z 1108.725,A -85,B 0,C 180,E1 15056.593,E2 15056.593} C_VEL
LIN {X 0,Y 420.595,Z 1121.901,A -85,B 0,C 180,E1 15053.837,E2 15053.837} C_VEL
LIN {X 0,Y 418.928,Z 1133.373,A -85,B 0,C 180,E1 15050.978,E2 15050.978} C_VEL
LIN {X 0,Y 417.672,Z 1143.602,A -85,B 0,C 180,E1 15047.988,E2 15047.988} C_VEL
LIN {X 0,Y 416.912,Z 1150.788,A -85,B 0,C 180,E1 15045.402,E2 15045.402} C_VEL
LIN {X 0,Y 416.345,Z 1157.771,A -85,B 0,C 180,E1 15042.341,E2 15042.341} C_VEL
LIN {X 0,Y 416.058,Z 1163.049,A -85,B 0,C 180,E1 15039.266,E2 15039.266} C_VEL
LIN {X 0,Y 415.939,Z 1166.757,A -85,B 0,C 180,E1 15036.349,E2 15036.349} C_VEL
LIN {X 0,Y 415.887,Z 1169.052,A -85,B 0,C 180,E1 15033.308,E2 15033.308} C_VEL
LIN {X 0,Y 415.885,Z 1169.893,A -85,B 0,C 180,E1 15030.689,E2 15030.689} C_VEL
LIN {X 0,Y 415.908,Z 1169.46,A -85,B 0,C 180,E1 15027.52,E2 15027.52} C_VEL
LIN {X 0,Y 415.918,Z 1167.726,A -85,B 0,C 180,E1 15024.759,E2 15024.759} C_VEL
LIN {X 0,Y 416.007,Z 1164.494,A -85,B 0,C 180,E1 15021.709,E2 15021.709} C_VEL
LIN {X 0,Y 416.226,Z 1159.572,A -85,B 0,C 180,E1 15018.64,E2 15018.64} C_VEL
LIN {X 0,Y 416.691,Z 1153.167,A -85,B 0,C 180,E1 15015.549,E2 15015.549} C_VEL
LIN {X 0,Y 417.379,Z 1146.114,A -85,B 0,C 180,E1 15012.863,E2 15012.863} C_VEL
LIN {X 0,Y 418.447,Z 1137.052,A -85,B 0,C 180,E1 15010.02,E2 15010.02} C_VEL
LIN {X 0,Y 419.955,Z 1125.953,A -85,B 0,C 180,E1 15007.13,E2 15007.13} C_VEL
LIN {X 0,Y 421.935,Z 1113.274,A -85,B 0,C 180,E1 15004.3,E2 15004.3} C_VEL
LIN {X 0,Y 424.194,Z 1099.644,A -85,B 0,C 180,E1 15001.72,E2 15001.72} C_VEL
LIN {X 0,Y 426.968,Z 1083.55,A -85,B 0,C 180,E1 14999.1,E2 14999.1} C_VEL
LIN {X 0,Y 429.793,Z 1067.535,A -85,B 0,C 180,E1 14996.859,E2 14996.859} C_VEL
LIN {X 0,Y 432.976,Z 1049.175,A -85,B 0,C 180,E1 14994.649,E2 14994.649} C_VEL
LIN {X 0,Y 436.194,Z 1030.344,A -85,B 0,C 180,E1 14992.693,E2 14992.693} C_VEL
LIN {X 0,Y 439.438,Z 1010.402,A -85,B 0,C 180,E1 14990.93,E2 14990.93} C_VEL
LIN {X 0,Y 442.732,Z 989.033,A -85,B 0,C 180,E1 14989.315,E2 14989.315} C_VEL
LIN {X 0,Y 445.571,Z 968.675,A -85,B 0,C 180,E1 14988.032,E2 14988.032} C_VEL
LIN {X 0,Y 448.365,Z 946.283,A -85,B 0,C 180,E1 14986.882,E2 14986.882} C_VEL
LIN {X 0,Y 450.603,Z 925.044,A -85,B 0,C 180,E1 14986.01,E2 14986.01} C_VEL
LIN {X 0,Y 452.492,Z 902.179,A -85,B 0,C 180,E1 14985.308,E2 14985.308} C_VEL
LIN {X 0,Y 453.794,Z 878.64,A -85,B 0,C 180,E1 14984.785,E2 14984.785} C_VEL
LIN {X 0,Y 461.201,Z 666.908,A -85,B 0,C 180,E1 14980.882,E2 14980.882} C_VEL
LIN {X 0,Y 463.488,Z 600.626,A -85,B 0,C 180,E1 14979.643,E2 14979.643} C_VEL
LIN {X 0,Y 451.52,Z 582.531,A -85,B 0,C 180,E1 14977.494,E2 14977.494} C_VEL
LIN {X 0,Y 440.16,Z 566.464,A -85,B 0,C 180,E1 14975.278,E2 14975.278} C_VEL
LIN {X 0,Y 431.269,Z 555.017,A -85,B 0,C 180,E1 14973.409,E2 14973.409} C_VEL
LIN {X 0,Y 428.753,Z 551.212,A -85,B 0,C 180,E1 14972.753,E2 14972.753} C_VEL
LIN {X 0,Y 425.263,Z 545.388,A -85,B 0,C 180,E1 14971.305,E2 14971.305} C_VEL
LIN {X 0,Y 422.918,Z 541.11,A -85,B 0,C 180,E1 14970.236,E2 14970.236} C_VEL
LIN {X 0,Y 420.836,Z 537.711,A -85,B 0,C 180,E1 14969.303,E2 14969.303} C_VEL
LIN {X 0,Y 420.041,Z 536.115,A -85,B 0,C 180,E1 14968.895,E2 14968.895} C_VEL
LIN {X 0,Y 417.932,Z 533.13,A -85,B 0,C 180,E1 14967.963,E2 14967.963} C_VEL
LIN {X 0,Y 417.405,Z 531.238,A -85,B 0,C 180,E1 14967.427,E2 14967.427} C_VEL
LIN {X 0,Y 417.371,Z 531.032,A -85,B 0,C 180,E1 14963.582,E2 14963.582} C_VEL
LIN {X 0,Y 417.369,Z 531.03,A -85,B 0,C 180,E1 14959.698,E2 14959.698} C_VEL
LIN {X 0,Y 417.372,Z 530.998,A -85,B 0,C 180,E1 14955.848,E2 14955.848} C_VEL
LIN {X 0,Y 417.37,Z 531.057,A -85,B 0,C 180,E1 14952.029,E2 14952.029} C_VEL
LIN {X 0,Y 417.362,Z 530.996,A -85,B 0,C 180,E1 14948.125,E2 14948.125} C_VEL
LIN {X 0,Y 417.373,Z 531.048,A -85,B 0,C 180,E1 14944.259,E2 14944.259} C_VEL
LIN {X 0,Y 417.373,Z 531.047,A -85,B 0,C 180,E1 14940.411,E2 14940.411} C_VEL
LIN {X 0,Y 417.372,Z 531.045,A -85,B 0,C 180,E1 14936.566,E2 14936.566} C_VEL
LIN {X 0,Y 417.381,Z 531.041,A -85,B 0,C 180,E1 14932.642,E2 14932.642} C_VEL
LIN {X 0,Y 417.361,Z 531.013,A -85,B 0,C 180,E1 14928.81,E2 14928.81} C_VEL
LIN {X 0,Y 417.364,Z 531.045,A -85,B 0,C 180,E1 14924.863,E2 14924.863} C_VEL
LIN {X 0,Y 417.368,Z 530.999,A -85,B 0,C 180,E1 14920.985,E2 14920.985} C_VEL
LIN {X 0,Y 417.376,Z 531.052,A -85,B 0,C 180,E1 14917.164,E2 14917.164} C_VEL
LIN {X 0,Y 417.373,Z 531.017,A -85,B 0,C 180,E1 14913.232,E2 14913.232} C_VEL
LIN {X 0,Y 417.402,Z 531.301,A -85,B 0,C 180,E1 14910.096,E2 14910.096} C_VEL
LIN {X 0,Y 418.874,Z 534.763,A -85,B 0,C 180,E1 14909.122,E2 14909.122} C_VEL
LIN {X 0,Y 420.437,Z 536.796,A -85,B 0,C 180,E1 14908.453,E2 14908.453} C_VEL
LIN {X 0,Y 422.337,Z 540.479,A -85,B 0,C 180,E1 14907.492,E2 14907.492} C_VEL
LIN {X 0,Y 423.544,Z 542.434,A -85,B 0,C 180,E1 14906.953,E2 14906.953} C_VEL
LIN {X 0,Y 426.5,Z 547.809,A -85,B 0,C 180,E1 14905.598,E2 14905.598} C_VEL
LIN {X 0,Y 431.222,Z 556.37,A -85,B 0,C 180,E1 14903.57,E2 14903.57} C_VEL
LIN {X 0,Y 437.686,Z 568.934,A -85,B 0,C 180,E1 14900.913,E2 14900.913} C_VEL
LIN {X 0,Y 444.452,Z 582.926,A -85,B 0,C 180,E1 14898.335,E2 14898.335} C_VEL
LIN {X 0,Y 455.594,Z 600.409,A -85,B 0,C 180,E1 14896.237,E2 14896.237} C_VEL
LIN {X 0,Y 459.299,Z 627.183,A -85,B 0,C 180,E1 14895.117,E2 14895.117} C_VEL
LIN {X 0,Y 452.647,Z 859.875,A -85,B 0,C 180,E1 14891.126,E2 14891.126} C_VEL
LIN {X 0,Y 451.377,Z 899.214,A -85,B 0,C 180,E1 14890.422,E2 14890.422} C_VEL
LIN {X 0,Y 450.46,Z 912.84,A -85,B 0,C 180,E1 14890.077,E2 14890.077} C_VEL
LIN {X 0,Y 448.962,Z 920.387,A -85,B 0,C 180,E1 14889.95,E2 14889.95} C_VEL
LIN {X 0,Y 442.999,Z 938.56,A -85,B 0,C 180,E1 14889.774,E2 14889.774} C_VEL
LIN {X 0,Y 441.327,Z 945.75,A -85,B 0,C 180,E1 14889.551,E2 14889.551} C_VEL
LIN {X 0,Y 441.191,Z 946.77,A -85,B 0,C 180,E1 14889.507,E2 14889.507} C_VEL
LIN {X 0,Y 438.408,Z 967.308,A -85,B 0,C 180,E1 14888.424,E2 14888.424} C_VEL
LIN {X 0,Y 435.4,Z 986.786,A -85,B 0,C 180,E1 14887.154,E2 14887.154} C_VEL
LIN {X 0,Y 432.069,Z 1005.34,A -85,B 0,C 180,E1 14885.673,E2 14885.673} C_VEL
LIN {X 0,Y 428.457,Z 1023.923,A -85,B 0,C 180,E1 14883.9,E2 14883.9} C_VEL
LIN {X 0,Y 424.906,Z 1041.309,A -85,B 0,C 180,E1 14881.928,E2 14881.928} C_VEL
LIN {X 0,Y 421.495,Z 1057.053,A -85,B 0,C 180,E1 14879.8,E2 14879.8} C_VEL
LIN {X 0,Y 418.338,Z 1071.724,A -85,B 0,C 180,E1 14877.47,E2 14877.47} C_VEL
LIN {X 0,Y 415.594,Z 1084.731,A -85,B 0,C 180,E1 14875.051,E2 14875.051} C_VEL
LIN {X 0,Y 413.123,Z 1096.989,A -85,B 0,C 180,E1 14872.332,E2 14872.332} C_VEL
LIN {X 0,Y 411.077,Z 1108.46,A -85,B 0,C 180,E1 14869.312,E2 14869.312} C_VEL
LIN {X 0,Y 409.673,Z 1117.947,A -85,B 0,C 180,E1 14866.3,E2 14866.3} C_VEL
LIN {X 0,Y 408.771,Z 1125.611,A -85,B 0,C 180,E1 14863.293,E2 14863.293} C_VEL
LIN {X 0,Y 408.251,Z 1131.599,A -85,B 0,C 180,E1 14860.299,E2 14860.299} C_VEL
LIN {X 0,Y 408.011,Z 1136.091,A -85,B 0,C 180,E1 14857.321,E2 14857.321} C_VEL
LIN {X 0,Y 407.933,Z 1138.954,A -85,B 0,C 180,E1 14854.358,E2 14854.358} C_VEL
LIN {X 0,Y 407.915,Z 1140.438,A -85,B 0,C 180,E1 14851.264,E2 14851.264} C_VEL
LIN {X 0,Y 407.913,Z 1140.409,A -85,B 0,C 180,E1 14848.455,E2 14848.455} C_VEL
LIN {X 0,Y 407.937,Z 1138.914,A -85,B 0,C 180,E1 14845.501,E2 14845.501} C_VEL
LIN {X 0,Y 408.013,Z 1136.033,A -85,B 0,C 180,E1 14842.537,E2 14842.537} C_VEL
LIN {X 0,Y 408.258,Z 1131.501,A -85,B 0,C 180,E1 14839.558,E2 14839.558} C_VEL
LIN {X 0,Y 408.818,Z 1125.139,A -85,B 0,C 180,E1 14836.421,E2 14836.421} C_VEL
LIN {X 0,Y 409.758,Z 1117.408,A -85,B 0,C 180,E1 14833.412,E2 14833.412} C_VEL
LIN {X 0,Y 411.198,Z 1107.747,A -85,B 0,C 180,E1 14830.393,E2 14830.393} C_VEL
LIN {X 0,Y 413.167,Z 1096.736,A -85,B 0,C 180,E1 14827.52,E2 14827.52} C_VEL
LIN {X 0,Y 415.653,Z 1084.435,A -85,B 0,C 180,E1 14824.8,E2 14824.8} C_VEL
LIN {X 0,Y 418.413,Z 1071.389,A -85,B 0,C 180,E1 14822.381,E2 14822.381} C_VEL
LIN {X 0,Y 421.691,Z 1056.153,A -85,B 0,C 180,E1 14819.98,E2 14819.98} C_VEL
LIN {X 0,Y 425.125,Z 1040.286,A -85,B 0,C 180,E1 14817.854,E2 14817.854} C_VEL
LIN {X 0,Y 428.701,Z 1022.803,A -85,B 0,C 180,E1 14815.891,E2 14815.891} C_VEL
LIN {X 0,Y 432.202,Z 1004.655,A -85,B 0,C 180,E1 14814.176,E2 14814.176} C_VEL
LIN {X 0,Y 435.546,Z 985.979,A -85,B 0,C 180,E1 14812.695,E2 14812.695} C_VEL
LIN {X 0,Y 438.5,Z 966.791,A -85,B 0,C 180,E1 14811.454,E2 14811.454} C_VEL
LIN {X 0,Y 441.368,Z 945.382,A -85,B 0,C 180,E1 14810.339,E2 14810.339} C_VEL
LIN {X 0,Y 443.619,Z 924.721,A -85,B 0,C 180,E1 14809.504,E2 14809.504} C_VEL
LIN {X 0,Y 445.267,Z 903.596,A -85,B 0,C 180,E1 14808.889,E2 14808.889} C_VEL
LIN {X 0,Y 446.459,Z 876.147,A -85,B 0,C 180,E1 14808.35,E2 14808.35} C_VEL
LIN {X 0,Y 453.153,Z 651.617,A -85,B 0,C 180,E1 14804.47,E2 14804.47} C_VEL
LIN {X 0,Y 453.634,Z 632.584,A -85,B 0,C 180,E1 14804.111,E2 14804.111} C_VEL
LIN {X 0,Y 448.591,Z 605.263,A -85,B 0,C 180,E1 14802.742,E2 14802.742} C_VEL
LIN {X 0,Y 437.939,Z 588.34,A -85,B 0,C 180,E1 14800.637,E2 14800.637} C_VEL
LIN {X 0,Y 433.62,Z 582.055,A -85,B 0,C 180,E1 14799.697,E2 14799.697} C_VEL
LIN {X 0,Y 430.27,Z 582.012,A -85,B 0,C 180,E1 14799.118,E2 14799.118} C_VEL
LIN {X 0,Y 427.586,Z 583.496,A -85,B 0,C 180,E1 14798.635,E2 14798.635} C_VEL
LIN {X 0,Y 426.873,Z 585.95,A -85,B 0,C 180,E1 14798.283,E2 14798.283} C_VEL
LIN {X 0,Y 424.752,Z 629.206,A -85,B 0,C 180,E1 14794.481,E2 14794.481} C_VEL
LIN {X 0,Y 422.63,Z 672.479,A -85,B 0,C 180,E1 14790.732,E2 14790.732} C_VEL
LIN {X 0,Y 420.47,Z 716.046,A -85,B 0,C 180,E1 14786.959,E2 14786.959} C_VEL
LIN {X 0,Y 420.354,Z 721.545,A -85,B 0,C 180,E1 14786.535,E2 14786.535} C_VEL
LIN {X 0,Y 421.111,Z 730.247,A -85,B 0,C 180,E1 14786.305,E2 14786.305} C_VEL
LIN {X 0,Y 417.623,Z 893.262,A -85,B 0,C 180,E1 14783.127,E2 14783.127} C_VEL
LIN {X 0,Y 417.172,Z 910.953,A -85,B 0,C 180,E1 14782.524,E2 14782.524} C_VEL
LIN {X 0,Y 416.42,Z 929.042,A -85,B 0,C 180,E1 14781.628,E2 14781.628} C_VEL
LIN {X 0,Y 415.558,Z 945.102,A -85,B 0,C 180,E1 14780.566,E2 14780.566} C_VEL
LIN {X 0,Y 414.514,Z 960.786,A -85,B 0,C 180,E1 14779.23,E2 14779.23} C_VEL
LIN {X 0,Y 413.433,Z 975.547,A -85,B 0,C 180,E1 14777.661,E2 14777.661} C_VEL
LIN {X 0,Y 412.452,Z 987.905,A -85,B 0,C 180,E1 14776.043,E2 14776.043} C_VEL
LIN {X 0,Y 411.507,Z 999.39,A -85,B 0,C 180,E1 14774.193,E2 14774.193} C_VEL
LIN {X 0,Y 410.688,Z 1009.966,A -85,B 0,C 180,E1 14772.086,E2 14772.086} C_VEL
LIN {X 0,Y 410.084,Z 1018.403,A -85,B 0,C 180,E1 14769.969,E2 14769.969} C_VEL
LIN {X 0,Y 409.646,Z 1025.312,A -85,B 0,C 180,E1 14767.708,E2 14767.708} C_VEL
LIN {X 0,Y 409.4,Z 1030.652,A -85,B 0,C 180,E1 14765.325,E2 14765.325} C_VEL
LIN {X 0,Y 409.309,Z 1034.132,A -85,B 0,C 180,E1 14762.941,E2 14762.941} C_VEL
LIN {X 0,Y 409.318,Z 1035.81,A -85,B 0,C 180,E1 14760.56,E2 14760.56} C_VEL
LIN {X 0,Y 409.402,Z 1035.8,A -85,B 0,C 180,E1 14758.181,E2 14758.181} C_VEL
LIN {X 0,Y 409.584,Z 1034.049,A -85,B 0,C 180,E1 14755.801,E2 14755.801} C_VEL
LIN {X 0,Y 409.888,Z 1030.411,A -85,B 0,C 180,E1 14753.417,E2 14753.417} C_VEL
LIN {X 0,Y 410.35,Z 1025.219,A -85,B 0,C 180,E1 14751.17,E2 14751.17} C_VEL
LIN {X 0,Y 410.96,Z 1018.576,A -85,B 0,C 180,E1 14749.061,E2 14749.061} C_VEL
LIN {X 0,Y 411.676,Z 1010.515,A -85,B 0,C 180,E1 14747.089,E2 14747.089} C_VEL
LIN {X 0,Y 412.575,Z 1000.286,A -85,B 0,C 180,E1 14745.115,E2 14745.115} C_VEL
LIN {X 0,Y 413.547,Z 988.907,A -85,B 0,C 180,E1 14743.352,E2 14743.352} C_VEL
LIN {X 0,Y 414.5,Z 976.437,A -85,B 0,C 180,E1 14741.798,E2 14741.798} C_VEL
LIN {X 0,Y 415.4,Z 962.2,A -85,B 0,C 180,E1 14740.381,E2 14740.381} C_VEL
LIN {X 0,Y 416.203,Z 946.931,A -85,B 0,C 180,E1 14739.174,E2 14739.174} C_VEL
LIN {X 0,Y 416.809,Z 930.948,A -85,B 0,C 180,E1 14738.21,E2 14738.21} C_VEL
LIN {X 0,Y 417.221,Z 913.102,A -85,B 0,C 180,E1 14737.431,E2 14737.431} C_VEL
LIN {X 0,Y 417.357,Z 895.111,A -85,B 0,C 180,E1 14736.921,E2 14736.921} C_VEL
LIN {X 0,Y 419.227,Z 805.906,A -85,B 0,C 180,E1 14735.106,E2 14735.106} C_VEL
LIN {X 0,Y 421.653,Z 737.071,A -85,B 0,C 180,E1 14733.564,E2 14733.564} C_VEL
LIN {X 0,Y 423.202,Z 728.951,A -85,B 0,C 180,E1 14733.024,E2 14733.024} C_VEL
LIN {X 0,Y 424.731,Z 685.969,A -85,B 0,C 180,E1 14729.542,E2 14729.542} C_VEL
LIN {X 0,Y 425.999,Z 641.326,A -85,B 0,C 180,E1 14726.041,E2 14726.041} C_VEL
LIN {X 0,Y 426.375,Z 633.726,A -85,B 0,C 180,E1 14725.425,E2 14725.425} C_VEL
LIN {X 0,Y 427.497,Z 631.93,A -85,B 0,C 180,E1 14725.121,E2 14725.121} C_VEL
LIN {X 0,Y 430.421,Z 629.22,A -85,B 0,C 180,E1 14724.681,E2 14724.681} C_VEL
LIN {X 0,Y 434.387,Z 622.975,A -85,B 0,C 180,E1 14724.182,E2 14724.182} C_VEL
LIN {X 0,Y 435.695,Z 620.843,A -85,B 0,C 180,E1 14724.022,E2 14724.022} C_VEL
LIN {X 0,Y 439.402,Z 617.548,A -85,B 0,C 180,E1 14723.505,E2 14723.505} C_VEL
LIN {X 0,Y 443.584,Z 611.502,A -85,B 0,C 180,E1 14722.999,E2 14722.999} C_VEL
LIN {X 0,Y 445.096,Z 609.173,A -85,B 0,C 180,E1 14722.824,E2 14722.824} C_VEL
LIN {X 0,Y 449.546,Z 604.896,A -85,B 0,C 180,E1 14722.252,E2 14722.252} C_VEL
LIN {X 0,Y 453.693,Z 599.173,A -85,B 0,C 180,E1 14721.778,E2 14721.778} C_VEL
LIN {X 0,Y 458.005,Z 606.221,A -85,B 0,C 180,E1 14720.987,E2 14720.987} C_VEL
LIN {X 0,Y 450.177,Z 815.575,A -85,B 0,C 180,E1 14717.081,E2 14717.081} C_VEL
LIN {X 0,Y 447.205,Z 893.222,A -85,B 0,C 180,E1 14715.61,E2 14715.61} C_VEL
LIN {X 0,Y 445.35,Z 916.422,A -85,B 0,C 180,E1 14714.969,E2 14714.969} C_VEL
LIN {X 0,Y 443.009,Z 939.765,A -85,B 0,C 180,E1 14714.089,E2 14714.089} C_VEL
LIN {X 0,Y 440.562,Z 959.563,A -85,B 0,C 180,E1 14713.133,E2 14713.133} C_VEL
LIN {X 0,Y 437.437,Z 981.663,A -85,B 0,C 180,E1 14711.829,E2 14711.829} C_VEL
LIN {X 0,Y 434.282,Z 1001.564,A -85,B 0,C 180,E1 14710.41,E2 14710.41} C_VEL
LIN {X 0,Y 430.716,Z 1022.391,A -85,B 0,C 180,E1 14708.642,E2 14708.642} C_VEL
LIN {X 0,Y 427.263,Z 1041.853,A -85,B 0,C 180,E1 14706.709,E2 14706.709} C_VEL
LIN {X 0,Y 423.618,Z 1061.425,A -85,B 0,C 180,E1 14704.424,E2 14704.424} C_VEL
LIN {X 0,Y 420.379,Z 1079.014,A -85,B 0,C 180,E1 14702.033,E2 14702.033} C_VEL
LIN {X 0,Y 417.657,Z 1093.849,A -85,B 0,C 180,E1 14699.706,E2 14699.706} C_VEL
LIN {X 0,Y 415.102,Z 1108.234,A -85,B 0,C 180,E1 14697.081,E2 14697.081} C_VEL
LIN {X 0,Y 413.025,Z 1120.683,A -85,B 0,C 180,E1 14694.454,E2 14694.454} C_VEL
LIN {X 0,Y 411.222,Z 1132.346,A -85,B 0,C 180,E1 14691.54,E2 14691.54} C_VEL
LIN {X 0,Y 409.914,Z 1142.296,A -85,B 0,C 180,E1 14688.635,E2 14688.635} C_VEL
LIN {X 0,Y 408.958,Z 1150.844,A -85,B 0,C 180,E1 14685.575,E2 14685.575} C_VEL
LIN {X 0,Y 408.366,Z 1158.016,A -85,B 0,C 180,E1 14682.443,E2 14682.443} C_VEL
LIN {X 0,Y 408.066,Z 1163.049,A -85,B 0,C 180,E1 14679.449,E2 14679.449} C_VEL
LIN {X 0,Y 407.946,Z 1166.757,A -85,B 0,C 180,E1 14676.474,E2 14676.474} C_VEL
LIN {X 0,Y 407.888,Z 1169.051,A -85,B 0,C 180,E1 14673.373,E2 14673.373} C_VEL
LIN {X 0,Y 407.885,Z 1169.893,A -85,B 0,C 180,E1 14670.702,E2 14670.702} C_VEL
LIN {X 0,Y 407.905,Z 1169.459,A -85,B 0,C 180,E1 14667.471,E2 14667.471} C_VEL
LIN {X 0,Y 407.917,Z 1167.726,A -85,B 0,C 180,E1 14664.656,E2 14664.656} C_VEL
LIN {X 0,Y 408.017,Z 1164.494,A -85,B 0,C 180,E1 14661.545,E2 14661.545} C_VEL
LIN {X 0,Y 408.241,Z 1159.827,A -85,B 0,C 180,E1 14658.557,E2 14658.557} C_VEL
LIN {X 0,Y 408.674,Z 1153.903,A -85,B 0,C 180,E1 14655.66,E2 14655.66} C_VEL
LIN {X 0,Y 409.443,Z 1146.114,A -85,B 0,C 180,E1 14652.667,E2 14652.667} C_VEL
LIN {X 0,Y 410.568,Z 1137.067,A -85,B 0,C 180,E1 14649.768,E2 14649.768} C_VEL
LIN {X 0,Y 412.145,Z 1126.106,A -85,B 0,C 180,E1 14646.844,E2 14646.844} C_VEL
LIN {X 0,Y 414.126,Z 1114.063,A -85,B 0,C 180,E1 14644.087,E2 14644.087} C_VEL
LIN {X 0,Y 416.47,Z 1100.497,A -85,B 0,C 180,E1 14641.461,E2 14641.461} C_VEL
LIN {X 0,Y 419.311,Z 1084.883,A -85,B 0,C 180,E1 14638.839,E2 14638.839} C_VEL
LIN {X 0,Y 422.293,Z 1068.682,A -85,B 0,C 180,E1 14636.518,E2 14636.518} C_VEL
LIN {X 0,Y 425.905,Z 1048.956,A -85,B 0,C 180,E1 14634.088,E2 14634.088} C_VEL
LIN {X 0,Y 429.483,Z 1029.591,A -85,B 0,C 180,E1 14632.033,E2 14632.033} C_VEL
LIN {X 0,Y 432.953,Z 1009.499,A -85,B 0,C 180,E1 14630.23,E2 14630.23} C_VEL
LIN {X 0,Y 436.539,Z 987.357,A -85,B 0,C 180,E1 14628.552,E2 14628.552} C_VEL
LIN {X 0,Y 439.632,Z 966.48,A -85,B 0,C 180,E1 14627.241,E2 14627.241} C_VEL
LIN {X 0,Y 442.433,Z 944.559,A -85,B 0,C 180,E1 14626.129,E2 14626.129} C_VEL
LIN {X 0,Y 444.836,Z 922.637,A -85,B 0,C 180,E1 14625.238,E2 14625.238} C_VEL
LIN {X 0,Y 446.693,Z 900.195,A -85,B 0,C 180,E1 14624.567,E2 14624.567} C_VEL
LIN {X 0,Y 448.101,Z 873.277,A -85,B 0,C 180,E1 14623.992,E2 14623.992} C_VEL
LIN {X 0,Y 455.866,Z 662.969,A -85,B 0,C 180,E1 14620.076,E2 14620.076} C_VEL
LIN {X 0,Y 457.948,Z 604.294,A -85,B 0,C 180,E1 14618.961,E2 14618.961} C_VEL
LIN {X 0,Y 445.69,Z 585.677,A -85,B 0,C 180,E1 14616.677,E2 14616.677} C_VEL
LIN {X 0,Y 433.29,Z 568.336,A -85,B 0,C 180,E1 14614.147,E2 14614.147} C_VEL
LIN {X 0,Y 424.265,Z 556.814,A -85,B 0,C 180,E1 14612.142,E2 14612.142} C_VEL
LIN {X 0,Y 421.097,Z 552.417,A -85,B 0,C 180,E1 14611.331,E2 14611.331} C_VEL
LIN {X 0,Y 417.73,Z 546.869,A -85,B 0,C 180,E1 14609.858,E2 14609.858} C_VEL
LIN {X 0,Y 415.219,Z 542.309,A -85,B 0,C 180,E1 14608.632,E2 14608.632} C_VEL
LIN {X 0,Y 412.96,Z 538.678,A -85,B 0,C 180,E1 14607.545,E2 14607.545} C_VEL
LIN {X 0,Y 412.019,Z 536.988,A -85,B 0,C 180,E1 14607.049,E2 14607.049} C_VEL
LIN {X 0,Y 409.947,Z 534.011,A -85,B 0,C 180,E1 14606.041,E2 14606.041} C_VEL
LIN {X 0,Y 409.465,Z 532.249,A -85,B 0,C 180,E1 14605.491,E2 14605.491} C_VEL
LIN {X 0,Y 409.426,Z 531.988,A -85,B 0,C 180,E1 14601.639,E2 14601.639} C_VEL
LIN {X 0,Y 409.433,Z 532.028,A -85,B 0,C 180,E1 14597.748,E2 14597.748} C_VEL
LIN {X 0,Y 409.435,Z 531.998,A -85,B 0,C 180,E1 14593.846,E2 14593.846} C_VEL
LIN {X 0,Y 409.425,Z 531.994,A -85,B 0,C 180,E1 14589.985,E2 14589.985} C_VEL
LIN {X 0,Y 409.43,Z 532.032,A -85,B 0,C 180,E1 14586.027,E2 14586.027} C_VEL
LIN {X 0,Y 409.435,Z 532.041,A -85,B 0,C 180,E1 14582.099,E2 14582.099} C_VEL
LIN {X 0,Y 409.435,Z 532.046,A -85,B 0,C 180,E1 14578.18,E2 14578.18} C_VEL
LIN {X 0,Y 409.435,Z 532.049,A -85,B 0,C 180,E1 14574.253,E2 14574.253} C_VEL
LIN {X 0,Y 409.438,Z 532.041,A -85,B 0,C 180,E1 14570.299,E2 14570.299} C_VEL
LIN {X 0,Y 409.433,Z 531.99,A -85,B 0,C 180,E1 14566.297,E2 14566.297} C_VEL
LIN {X 0,Y 409.422,Z 532.01,A -85,B 0,C 180,E1 14562.519,E2 14562.519} C_VEL
LIN {X 0,Y 409.424,Z 532.024,A -85,B 0,C 180,E1 14558.505,E2 14558.505} C_VEL
LIN {X 0,Y 409.429,Z 531.989,A -85,B 0,C 180,E1 14554.632,E2 14554.632} C_VEL
LIN {X 0,Y 409.459,Z 532.278,A -85,B 0,C 180,E1 14552.04,E2 14552.04} C_VEL
LIN {X 0,Y 411.082,Z 535.969,A -85,B 0,C 180,E1 14550.892,E2 14550.892} C_VEL
LIN {X 0,Y 412.641,Z 538.012,A -85,B 0,C 180,E1 14550.165,E2 14550.165} C_VEL
LIN {X 0,Y 414.662,Z 541.716,A -85,B 0,C 180,E1 14549.096,E2 14549.096} C_VEL
LIN {X 0,Y 415.797,Z 543.583,A -85,B 0,C 180,E1 14548.546,E2 14548.546} C_VEL
LIN {X 0,Y 418.641,Z 548.602,A -85,B 0,C 180,E1 14547.169,E2 14547.169} C_VEL
LIN {X 0,Y 423.721,Z 557.803,A -85,B 0,C 180,E1 14544.846,E2 14544.846} C_VEL
LIN {X 0,Y 430.455,Z 570.795,A -85,B 0,C 180,E1 14541.946,E2 14541.946} C_VEL
LIN {X 0,Y 436.135,Z 582.212,A -85,B 0,C 180,E1 14539.722,E2 14539.722} C_VEL
LIN {X 0,Y 448.846,Z 601.789,A -85,B 0,C 180,E1 14537.201,E2 14537.201} C_VEL
LIN {X 0,Y 450.764,Z 605.356,A -85,B 0,C 180,E1 14536.83,E2 14536.83} C_VEL
LIN {X 0,Y 453.883,Z 628.866,A -85,B 0,C 180,E1 14535.837,E2 14535.837} C_VEL
LIN {X 0,Y 446.861,Z 860.923,A -85,B 0,C 180,E1 14531.819,E2 14531.819} C_VEL
LIN {X 0,Y 445.54,Z 899.377,A -85,B 0,C 180,E1 14531.123,E2 14531.123} C_VEL
LIN {X 0,Y 443.948,Z 920.429,A -85,B 0,C 180,E1 14530.545,E2 14530.545} C_VEL
LIN {X 0,Y 441.816,Z 941.511,A -85,B 0,C 180,E1 14529.741,E2 14529.741} C_VEL
LIN {X 0,Y 441.191,Z 946.77,A -85,B 0,C 180,E1 14529.507,E2 14529.507} C_VEL
LIN {X 0,Y 439.54,Z 954.094,A -85,B 0,C 180,E1 14529.246,E2 14529.246} C_VEL
LIN {X 0,Y 432.324,Z 972.478,A -85,B 0,C 180,E1 14528.732,E2 14528.732} C_VEL
LIN {X 0,Y 430.409,Z 979.412,A -85,B 0,C 180,E1 14528.364,E2 14528.364} C_VEL
LIN {X 0,Y 427.117,Z 998.088,A -85,B 0,C 180,E1 14526.986,E2 14526.986} C_VEL
LIN {X 0,Y 423.499,Z 1016.38,A -85,B 0,C 180,E1 14525.341,E2 14525.341} C_VEL
LIN {X 0,Y 419.636,Z 1034.569,A -85,B 0,C 180,E1 14523.395,E2 14523.395} C_VEL
LIN {X 0,Y 416.066,Z 1050.746,A -85,B 0,C 180,E1 14521.351,E2 14521.351} C_VEL
LIN {X 0,Y 412.682,Z 1065.447,A -85,B 0,C 180,E1 14519.143,E2 14519.143} C_VEL
LIN {X 0,Y 409.357,Z 1080.16,A -85,B 0,C 180,E1 14516.55,E2 14516.55} C_VEL
LIN {X 0,Y 406.641,Z 1092.738,A -85,B 0,C 180,E1 14513.935,E2 14513.935} C_VEL
LIN {X 0,Y 404.36,Z 1103.841,A -85,B 0,C 180,E1 14511.162,E2 14511.162} C_VEL
LIN {X 0,Y 402.443,Z 1114.595,A -85,B 0,C 180,E1 14507.943,E2 14507.943} C_VEL
LIN {X 0,Y 401.238,Z 1122.987,A -85,B 0,C 180,E1 14504.873,E2 14504.873} C_VEL
LIN {X 0,Y 400.513,Z 1129.614,A -85,B 0,C 180,E1 14501.812,E2 14501.812} C_VEL
LIN {X 0,Y 400.121,Z 1134.86,A -85,B 0,C 180,E1 14498.623,E2 14498.623} C_VEL
LIN {X 0,Y 399.966,Z 1138.385,A -85,B 0,C 180,E1 14495.595,E2 14495.595} C_VEL
LIN {X 0,Y 399.916,Z 1140.316,A -85,B 0,C 180,E1 14492.579,E2 14492.579} C_VEL
LIN {X 0,Y 399.912,Z 1140.853,A -85,B 0,C 180,E1 14489.427,E2 14489.427} C_VEL
LIN {X 0,Y 399.927,Z 1139.964,A -85,B 0,C 180,E1 14486.56,E2 14486.56} C_VEL
LIN {X 0,Y 400.005,Z 1137.427,A -85,B 0,C 180,E1 14483.397,E2 14483.397} C_VEL
LIN {X 0,Y 400.203,Z 1133.571,A -85,B 0,C 180,E1 14480.364,E2 14480.364} C_VEL
LIN {X 0,Y 400.649,Z 1128.049,A -85,B 0,C 180,E1 14477.314,E2 14477.314} C_VEL
LIN {X 0,Y 401.551,Z 1120.581,A -85,B 0,C 180,E1 14474.103,E2 14474.103} C_VEL
LIN {X 0,Y 402.86,Z 1112.217,A -85,B 0,C 180,E1 14471.177,E2 14471.177} C_VEL
LIN {X 0,Y 404.725,Z 1101.981,A -85,B 0,C 180,E1 14468.249,E2 14468.249} C_VEL
LIN {X 0,Y 407.247,Z 1089.778,A -85,B 0,C 180,E1 14465.331,E2 14465.331} C_VEL
LIN {X 0,Y 410.129,Z 1076.824,A -85,B 0,C 180,E1 14462.721,E2 14462.721} C_VEL
LIN {X 0,Y 413.421,Z 1062.257,A -85,B 0,C 180,E1 14460.255,E2 14460.255} C_VEL
LIN {X 0,Y 416.987,Z 1046.523,A -85,B 0,C 180,E1 14458,E2 14458} C_VEL
LIN {X 0,Y 420.696,Z 1029.875,A -85,B 0,C 180,E1 14455.97,E2 14455.97} C_VEL
LIN {X 0,Y 424.213,Z 1012.886,A -85,B 0,C 180,E1 14454.23,E2 14454.23} C_VEL
LIN {X 0,Y 427.901,Z 993.794,A -85,B 0,C 180,E1 14452.589,E2 14452.589} C_VEL
LIN {X 0,Y 431.205,Z 974.908,A -85,B 0,C 180,E1 14451.239,E2 14451.239} C_VEL
LIN {X 0,Y 434.136,Z 955.148,A -85,B 0,C 180,E1 14450.102,E2 14450.102} C_VEL
LIN {X 0,Y 436.782,Z 933.683,A -85,B 0,C 180,E1 14449.119,E2 14449.119} C_VEL
LIN {X 0,Y 438.847,Z 912.539,A -85,B 0,C 180,E1 14448.398,E2 14448.398} C_VEL
LIN {X 0,Y 440.229,Z 890.752,A -85,B 0,C 180,E1 14447.888,E2 14447.888} C_VEL
LIN {X 0,Y 447.493,Z 661.482,A -85,B 0,C 180,E1 14443.882,E2 14443.882} C_VEL
LIN {X 0,Y 448.277,Z 634.31,A -85,B 0,C 180,E1 14443.372,E2 14443.372} C_VEL
LIN {X 0,Y 443.858,Z 609.9,A -85,B 0,C 180,E1 14442.124,E2 14442.124} C_VEL
LIN {X 0,Y 433.769,Z 593.784,A -85,B 0,C 180,E1 14440.068,E2 14440.068} C_VEL
LIN {X 0,Y 430.947,Z 589.866,A -85,B 0,C 180,E1 14439.474,E2 14439.474} C_VEL
LIN {X 0,Y 428.599,Z 591.003,A -85,B 0,C 180,E1 14439.084,E2 14439.084} C_VEL
LIN {X 0,Y 424.028,Z 598.057,A -85,B 0,C 180,E1 14438.435,E2 14438.435} C_VEL
LIN {X 0,Y 421.075,Z 600.809,A -85,B 0,C 180,E1 14437.953,E2 14437.953} C_VEL
LIN {X 0,Y 419.538,Z 601.922,A -85,B 0,C 180,E1 14437.598,E2 14437.598} C_VEL
LIN {X 0,Y 418.968,Z 604.858,A -85,B 0,C 180,E1 14437.227,E2 14437.227} C_VEL
LIN {X 0,Y 416.768,Z 647.265,A -85,B 0,C 180,E1 14433.49,E2 14433.49} C_VEL
LIN {X 0,Y 414.543,Z 690.437,A -85,B 0,C 180,E1 14429.713,E2 14429.713} C_VEL
LIN {X 0,Y 413.024,Z 722.304,A -85,B 0,C 180,E1 14426.975,E2 14426.975} C_VEL
LIN {X 0,Y 413.772,Z 731.137,A -85,B 0,C 180,E1 14426.734,E2 14426.734} C_VEL
LIN {X 0,Y 410.072,Z 894.339,A -85,B 0,C 180,E1 14423.475,E2 14423.475} C_VEL
LIN {X 0,Y 409.605,Z 912.044,A -85,B 0,C 180,E1 14422.861,E2 14422.861} C_VEL
LIN {X 0,Y 408.848,Z 929.733,A -85,B 0,C 180,E1 14421.973,E2 14421.973} C_VEL
LIN {X 0,Y 407.955,Z 945.939,A -85,B 0,C 180,E1 14420.892,E2 14420.892} C_VEL
LIN {X 0,Y 406.904,Z 961.273,A -85,B 0,C 180,E1 14419.577,E2 14419.577} C_VEL
LIN {X 0,Y 405.778,Z 976.137,A -85,B 0,C 180,E1 14417.986,E2 14417.986} C_VEL
LIN {X 0,Y 404.763,Z 988.543,A -85,B 0,C 180,E1 14416.356,E2 14416.356} C_VEL
LIN {X 0,Y 403.774,Z 1000.144,A -85,B 0,C 180,E1 14414.48,E2 14414.48} C_VEL
LIN {X 0,Y 402.901,Z 1010.913,A -85,B 0,C 180,E1 14412.323,E2 14412.323} C_VEL
LIN {X 0,Y 402.264,Z 1019.487,A -85,B 0,C 180,E1 14410.165,E2 14410.165} C_VEL
LIN {X 0,Y 401.796,Z 1026.477,A -85,B 0,C 180,E1 14407.867,E2 14407.867} C_VEL
LIN {X 0,Y 401.533,Z 1031.936,A -85,B 0,C 180,E1 14405.43,E2 14405.43} C_VEL
LIN {X 0,Y 401.439,Z 1035.352,A -85,B 0,C 180,E1 14403.141,E2 14403.141} C_VEL
LIN {X 0,Y 401.447,Z 1037.196,A -85,B 0,C 180,E1 14400.714,E2 14400.714} C_VEL
LIN {X 0,Y 401.536,Z 1037.322,A -85,B 0,C 180,E1 14398.288,E2 14398.288} C_VEL
LIN {X 0,Y 401.733,Z 1035.717,A -85,B 0,C 180,E1 14395.861,E2 14395.861} C_VEL
LIN {X 0,Y 402.044,Z 1032.508,A -85,B 0,C 180,E1 14393.575,E2 14393.575} C_VEL
LIN {X 0,Y 402.513,Z 1027.523,A -85,B 0,C 180,E1 14391.285,E2 14391.285} C_VEL
LIN {X 0,Y 403.194,Z 1020.598,A -85,B 0,C 180,E1 14388.992,E2 14388.992} C_VEL
LIN {X 0,Y 403.963,Z 1012.699,A -85,B 0,C 180,E1 14386.984,E2 14386.984} C_VEL
LIN {X 0,Y 404.907,Z 1002.604,A -85,B 0,C 180,E1 14384.973,E2 14384.973} C_VEL
LIN {X 0,Y 405.961,Z 990.812,A -85,B 0,C 180,E1 14383.105,E2 14383.105} C_VEL
LIN {X 0,Y 406.984,Z 978.183,A -85,B 0,C 180,E1 14381.498,E2 14381.498} C_VEL
LIN {X 0,Y 407.919,Z 964.244,A -85,B 0,C 180,E1 14380.081,E2 14380.081} C_VEL
LIN {X 0,Y 408.743,Z 948.962,A -85,B 0,C 180,E1 14378.85,E2 14378.85} C_VEL
LIN {X 0,Y 409.382,Z 933.109,A -85,B 0,C 180,E1 14377.869,E2 14377.869} C_VEL
LIN {X 0,Y 409.821,Z 915.262,A -85,B 0,C 180,E1 14377.066,E2 14377.066} C_VEL
LIN {X 0,Y 409.968,Z 897.471,A -85,B 0,C 180,E1 14376.543,E2 14376.543} C_VEL
LIN {X 0,Y 411.868,Z 813.356,A -85,B 0,C 180,E1 14374.765,E2 14374.765} C_VEL
LIN {X 0,Y 414.722,Z 739.496,A -85,B 0,C 180,E1 14373.048,E2 14373.048} C_VEL
LIN {X 0,Y 416.504,Z 730.714,A -85,B 0,C 180,E1 14372.477,E2 14372.477} C_VEL
LIN {X 0,Y 418.21,Z 687.08,A -85,B 0,C 180,E1 14368.909,E2 14368.909} C_VEL
LIN {X 0,Y 419.592,Z 652.395,A -85,B 0,C 180,E1 14366.11,E2 14366.11} C_VEL
LIN {X 0,Y 420.713,Z 650.585,A -85,B 0,C 180,E1 14365.802,E2 14365.802} C_VEL
LIN {X 0,Y 423.782,Z 647.553,A -85,B 0,C 180,E1 14365.327,E2 14365.327} C_VEL
LIN {X 0,Y 427.441,Z 641.659,A -85,B 0,C 180,E1 14364.85,E2 14364.85} C_VEL
LIN {X 0,Y 428.858,Z 639.093,A -85,B 0,C 180,E1 14364.677,E2 14364.677} C_VEL
LIN {X 0,Y 432.601,Z 635.763,A -85,B 0,C 180,E1 14364.133,E2 14364.133} C_VEL
LIN {X 0,Y 436.826,Z 629.646,A -85,B 0,C 180,E1 14363.602,E2 14363.602} C_VEL
LIN {X 0,Y 438.511,Z 627.041,A -85,B 0,C 180,E1 14363.399,E2 14363.399} C_VEL
LIN {X 0,Y 442.938,Z 622.581,A -85,B 0,C 180,E1 14362.815,E2 14362.815} C_VEL
LIN {X 0,Y 448.022,Z 615.249,A -85,B 0,C 180,E1 14362.222,E2 14362.222} C_VEL
LIN {X 0,Y 452.534,Z 610.933,A -85,B 0,C 180,E1 14361.659,E2 14361.659} C_VEL
LIN {X 0,Y 444.364,Z 819,A -85,B 0,C 180,E1 14357.742,E2 14357.742} C_VEL
LIN {X 0,Y 441.368,Z 893.331,A -85,B 0,C 180,E1 14356.318,E2 14356.318} C_VEL
LIN {X 0,Y 439.424,Z 916.566,A -85,B 0,C 180,E1 14355.671,E2 14355.671} C_VEL
LIN {X 0,Y 437.025,Z 939.447,A -85,B 0,C 180,E1 14354.803,E2 14354.803} C_VEL
LIN {X 0,Y 434.386,Z 959.842,A -85,B 0,C 180,E1 14353.809,E2 14353.809} C_VEL
LIN {X 0,Y 431.026,Z 982.389,A -85,B 0,C 180,E1 14352.457,E2 14352.457} C_VEL
LIN {X 0,Y 427.793,Z 1001.782,A -85,B 0,C 180,E1 14351.054,E2 14351.054} C_VEL
LIN {X 0,Y 424.051,Z 1022.392,A -85,B 0,C 180,E1 14349.279,E2 14349.279} C_VEL
LIN {X 0,Y 420.427,Z 1041.659,A -85,B 0,C 180,E1 14347.333,E2 14347.333} C_VEL
LIN {X 0,Y 416.764,Z 1059.959,A -85,B 0,C 180,E1 14345.155,E2 14345.155} C_VEL
LIN {X 0,Y 413.011,Z 1079.087,A -85,B 0,C 180,E1 14342.51,E2 14342.51} C_VEL
LIN {X 0,Y 409.993,Z 1094.799,A -85,B 0,C 180,E1 14339.996,E2 14339.996} C_VEL
LIN {X 0,Y 407.305,Z 1109.109,A -85,B 0,C 180,E1 14337.298,E2 14337.298} C_VEL
LIN {X 0,Y 405.069,Z 1121.989,A -85,B 0,C 180,E1 14334.5,E2 14334.5} C_VEL
LIN {X 0,Y 403.262,Z 1133.214,A -85,B 0,C 180,E1 14331.6,E2 14331.6} C_VEL
LIN {X 0,Y 401.832,Z 1143.579,A -85,B 0,C 180,E1 14328.422,E2 14328.422} C_VEL
LIN {X 0,Y 400.97,Z 1151.112,A -85,B 0,C 180,E1 14325.623,E2 14325.623} C_VEL
LIN {X 0,Y 400.36,Z 1158.188,A -85,B 0,C 180,E1 14322.403,E2 14322.403} C_VEL
LIN {X 0,Y 400.067,Z 1163.053,A -85,B 0,C 180,E1 14319.494,E2 14319.494} C_VEL
LIN {X 0,Y 399.945,Z 1166.834,A -85,B 0,C 180,E1 14316.459,E2 14316.459} C_VEL
LIN {X 0,Y 399.89,Z 1169.037,A -85,B 0,C 180,E1 14313.44,E2 14313.44} C_VEL
LIN {X 0,Y 399.888,Z 1169.87,A -85,B 0,C 180,E1 14310.86,E2 14310.86} C_VEL
LIN {X 0,Y 399.91,Z 1169.592,A -85,B 0,C 180,E1 14307.707,E2 14307.707} C_VEL
LIN {X 0,Y 399.917,Z 1167.789,A -85,B 0,C 180,E1 14304.692,E2 14304.692} C_VEL
LIN {X 0,Y 400.006,Z 1164.86,A -85,B 0,C 180,E1 14301.809,E2 14301.809} C_VEL
LIN {X 0,Y 400.235,Z 1160.033,A -85,B 0,C 180,E1 14298.618,E2 14298.618} C_VEL
LIN {X 0,Y 400.665,Z 1154.231,A -85,B 0,C 180,E1 14295.697,E2 14295.697} C_VEL
LIN {X 0,Y 401.512,Z 1146.113,A -85,B 0,C 180,E1 14292.463,E2 14292.463} C_VEL
LIN {X 0,Y 402.625,Z 1137.56,A -85,B 0,C 180,E1 14289.655,E2 14289.655} C_VEL
LIN {X 0,Y 404.349,Z 1126.204,A -85,B 0,C 180,E1 14286.54,E2 14286.54} C_VEL
LIN {X 0,Y 406.434,Z 1114.064,A -85,B 0,C 180,E1 14283.716,E2 14283.716} C_VEL
LIN {X 0,Y 408.903,Z 1100.537,A -85,B 0,C 180,E1 14281.043,E2 14281.043} C_VEL
LIN {X 0,Y 411.888,Z 1084.954,A -85,B 0,C 180,E1 14278.376,E2 14278.376} C_VEL
LIN {X 0,Y 415.24,Z 1067.751,A -85,B 0,C 180,E1 14275.872,E2 14275.872} C_VEL
LIN {X 0,Y 419.008,Z 1048.594,A -85,B 0,C 180,E1 14273.461,E2 14273.461} C_VEL
LIN {X 0,Y 422.633,Z 1030.183,A -85,B 0,C 180,E1 14271.468,E2 14271.468} C_VEL
LIN {X 0,Y 426.255,Z 1010.38,A -85,B 0,C 180,E1 14269.653,E2 14269.653} C_VEL
LIN {X 0,Y 429.857,Z 989.558,A -85,B 0,C 180,E1 14268.03,E2 14268.03} C_VEL
LIN {X 0,Y 433.043,Z 969.028,A -85,B 0,C 180,E1 14266.705,E2 14266.705} C_VEL
LIN {X 0,Y 436.193,Z 946.134,A -85,B 0,C 180,E1 14265.504,E2 14265.504} C_VEL
LIN {X 0,Y 438.567,Z 925.574,A -85,B 0,C 180,E1 14264.644,E2 14264.644} C_VEL
LIN {X 0,Y 440.68,Z 902.314,A -85,B 0,C 180,E1 14263.914,E2 14263.914} C_VEL
LIN {X 0,Y 442.102,Z 878.791,A -85,B 0,C 180,E1 14263.382,E2 14263.382} C_VEL
LIN {X 0,Y 450.27,Z 667.882,A -85,B 0,C 180,E1 14259.417,E2 14259.417} C_VEL
LIN {X 0,Y 452.538,Z 608.117,A -85,B 0,C 180,E1 14258.277,E2 14258.277} C_VEL
LIN {X 0,Y 440.949,Z 590.508,A -85,B 0,C 180,E1 14256.044,E2 14256.044} C_VEL
LIN {X 0,Y 429.658,Z 574.575,A -85,B 0,C 180,E1 14253.671,E2 14253.671} C_VEL
LIN {X 0,Y 421.01,Z 563.381,A -85,B 0,C 180,E1 14251.698,E2 14251.698} C_VEL
LIN {X 0,Y 417.088,Z 558.386,A -85,B 0,C 180,E1 14250.744,E2 14250.744} C_VEL
LIN {X 0,Y 413.256,Z 553.449,A -85,B 0,C 180,E1 14249.735,E2 14249.735} C_VEL
LIN {X 0,Y 410.407,Z 548.492,A -85,B 0,C 180,E1 14248.363,E2 14248.363} C_VEL
LIN {X 0,Y 408.161,Z 544.648,A -85,B 0,C 180,E1 14247.223,E2 14247.223} C_VEL
LIN {X 0,Y 405.059,Z 539.589,A -85,B 0,C 180,E1 14245.592,E2 14245.592} C_VEL
LIN {X 0,Y 404.335,Z 538.246,A -85,B 0,C 180,E1 14245.168,E2 14245.168} C_VEL
LIN {X 0,Y 401.983,Z 534.949,A -85,B 0,C 180,E1 14243.918,E2 14243.918} C_VEL
LIN {X 0,Y 401.527,Z 533.216,A -85,B 0,C 180,E1 14243.324,E2 14243.324} C_VEL
LIN {X 0,Y 401.491,Z 533.008,A -85,B 0,C 180,E1 14239.494,E2 14239.494} C_VEL
LIN {X 0,Y 401.488,Z 532.969,A -85,B 0,C 180,E1 14235.467,E2 14235.467} C_VEL
LIN {X 0,Y 401.496,Z 533.025,A -85,B 0,C 180,E1 14231.491,E2 14231.491} C_VEL
LIN {X 0,Y 401.5,Z 532.975,A -85,B 0,C 180,E1 14227.44,E2 14227.44} C_VEL
LIN {X 0,Y 401.49,Z 533.019,A -85,B 0,C 180,E1 14223.569,E2 14223.569} C_VEL
LIN {X 0,Y 401.489,Z 533.021,A -85,B 0,C 180,E1 14219.572,E2 14219.572} C_VEL
LIN {X 0,Y 401.491,Z 533.023,A -85,B 0,C 180,E1 14215.572,E2 14215.572} C_VEL
LIN {X 0,Y 401.5,Z 533.025,A -85,B 0,C 180,E1 14211.695,E2 14211.695} C_VEL
LIN {X 0,Y 401.489,Z 532.969,A -85,B 0,C 180,E1 14207.779,E2 14207.779} C_VEL
LIN {X 0,Y 401.499,Z 533.036,A -85,B 0,C 180,E1 14203.804,E2 14203.804} C_VEL
LIN {X 0,Y 401.494,Z 532.977,A -85,B 0,C 180,E1 14199.862,E2 14199.862} C_VEL
LIN {X 0,Y 401.483,Z 532.992,A -85,B 0,C 180,E1 14196.05,E2 14196.05} C_VEL
LIN {X 0,Y 401.528,Z 533.307,A -85,B 0,C 180,E1 14194.165,E2 14194.165} C_VEL
LIN {X 0,Y 403.284,Z 537.127,A -85,B 0,C 180,E1 14192.858,E2 14192.858} C_VEL
LIN {X 0,Y 404.712,Z 538.772,A -85,B 0,C 180,E1 14192.164,E2 14192.164} C_VEL
LIN {X 0,Y 406.591,Z 542.523,A -85,B 0,C 180,E1 14191.023,E2 14191.023} C_VEL
LIN {X 0,Y 407.991,Z 544.552,A -85,B 0,C 180,E1 14190.327,E2 14190.327} C_VEL
LIN {X 0,Y 410.953,Z 549.736,A -85,B 0,C 180,E1 14188.786,E2 14188.786} C_VEL
LIN {X 0,Y 414.014,Z 555.337,A -85,B 0,C 180,E1 14187.25,E2 14187.25} C_VEL
LIN {X 0,Y 418.49,Z 563.347,A -85,B 0,C 180,E1 14185.178,E2 14185.178} C_VEL
LIN {X 0,Y 425.298,Z 576.782,A -85,B 0,C 180,E1 14182.149,E2 14182.149} C_VEL
LIN {X 0,Y 427.782,Z 581.588,A -85,B 0,C 180,E1 14181.215,E2 14181.215} C_VEL
LIN {X 0,Y 437.971,Z 596.804,A -85,B 0,C 180,E1 14179.043,E2 14179.043} C_VEL
LIN {X 0,Y 445.872,Z 609.577,A -85,B 0,C 180,E1 14177.47,E2 14177.47} C_VEL
LIN {X 0,Y 448.542,Z 630.504,A -85,B 0,C 180,E1 14176.576,E2 14176.576} C_VEL
LIN {X 0,Y 441.103,Z 863.147,A -85,B 0,C 180,E1 14172.51,E2 14172.51} C_VEL
LIN {X 0,Y 439.756,Z 899.652,A -85,B 0,C 180,E1 14171.839,E2 14171.839} C_VEL
LIN {X 0,Y 438.082,Z 920.791,A -85,B 0,C 180,E1 14171.253,E2 14171.253} C_VEL
LIN {X 0,Y 435.834,Z 941.954,A -85,B 0,C 180,E1 14170.437,E2 14170.437} C_VEL
LIN {X 0,Y 433.272,Z 961.386,A -85,B 0,C 180,E1 14169.477,E2 14169.477} C_VEL
LIN {X 0,Y 430.409,Z 979.412,A -85,B 0,C 180,E1 14168.364,E2 14168.364} C_VEL
LIN {X 0,Y 428.476,Z 986.401,A -85,B 0,C 180,E1 14167.974,E2 14167.974} C_VEL
LIN {X 0,Y 420.573,Z 1003.768,A -85,B 0,C 180,E1 14167.136,E2 14167.136} C_VEL
LIN {X 0,Y 418.412,Z 1010.233,A -85,B 0,C 180,E1 14166.635,E2 14166.635} C_VEL
LIN {X 0,Y 414.587,Z 1027.727,A -85,B 0,C 180,E1 14164.86,E2 14164.86} C_VEL
LIN {X 0,Y 410.52,Z 1045.367,A -85,B 0,C 180,E1 14162.732,E2 14162.732} C_VEL
LIN {X 0,Y 406.914,Z 1060.577,A -85,B 0,C 180,E1 14160.573,E2 14160.573} C_VEL
LIN {X 0,Y 403.301,Z 1075.521,A -85,B 0,C 180,E1 14158.043,E2 14158.043} C_VEL
LIN {X 0,Y 400.072,Z 1089.197,A -85,B 0,C 180,E1 14155.3,E2 14155.3} C_VEL
LIN {X 0,Y 397.462,Z 1101.062,A -85,B 0,C 180,E1 14152.481,E2 14152.481} C_VEL
LIN {X 0,Y 395.367,Z 1111.474,A -85,B 0,C 180,E1 14149.501,E2 14149.501} C_VEL
LIN {X 0,Y 393.823,Z 1120.432,A -85,B 0,C 180,E1 14146.368,E2 14146.368} C_VEL
LIN {X 0,Y 392.803,Z 1127.988,A -85,B 0,C 180,E1 14143.094,E2 14143.094} C_VEL
LIN {X 0,Y 392.265,Z 1133.539,A -85,B 0,C 180,E1 14139.981,E2 14139.981} C_VEL
LIN {X 0,Y 392.026,Z 1137.656,A -85,B 0,C 180,E1 14136.738,E2 14136.738} C_VEL
LIN {X 0,Y 391.935,Z 1140.221,A -85,B 0,C 180,E1 14133.51,E2 14133.51} C_VEL
LIN {X 0,Y 391.919,Z 1141.13,A -85,B 0,C 180,E1 14130.585,E2 14130.585} C_VEL
LIN {X 0,Y 391.924,Z 1140.652,A -85,B 0,C 180,E1 14127.368,E2 14127.368} C_VEL
LIN {X 0,Y 391.967,Z 1138.869,A -85,B 0,C 180,E1 14124.437,E2 14124.437} C_VEL
LIN {X 0,Y 392.14,Z 1135.516,A -85,B 0,C 180,E1 14121.348,E2 14121.348} C_VEL
LIN {X 0,Y 392.527,Z 1130.759,A -85,B 0,C 180,E1 14118.242,E2 14118.242} C_VEL
LIN {X 0,Y 393.291,Z 1124.098,A -85,B 0,C 180,E1 14115.033,E2 14115.033} C_VEL
LIN {X 0,Y 394.579,Z 1115.783,A -85,B 0,C 180,E1 14111.839,E2 14111.839} C_VEL
LIN {X 0,Y 396.382,Z 1106.315,A -85,B 0,C 180,E1 14108.856,E2 14108.856} C_VEL
LIN {X 0,Y 398.68,Z 1095.415,A -85,B 0,C 180,E1 14106.028,E2 14106.028} C_VEL
LIN {X 0,Y 401.627,Z 1082.553,A -85,B 0,C 180,E1 14103.217,E2 14103.217} C_VEL
LIN {X 0,Y 404.981,Z 1068.598,A -85,B 0,C 180,E1 14100.636,E2 14100.636} C_VEL
LIN {X 0,Y 408.528,Z 1053.785,A -85,B 0,C 180,E1 14098.333,E2 14098.333} C_VEL
LIN {X 0,Y 412.487,Z 1036.97,A -85,B 0,C 180,E1 14096.116,E2 14096.116} C_VEL
LIN {X 0,Y 416.369,Z 1019.949,A -85,B 0,C 180,E1 14094.216,E2 14094.216} C_VEL
LIN {X 0,Y 420.068,Z 1002.003,A -85,B 0,C 180,E1 14092.544,E2 14092.544} C_VEL
LIN {X 0,Y 423.941,Z 981.593,A -85,B 0,C 180,E1 14090.971,E2 14090.971} C_VEL
LIN {X 0,Y 427.281,Z 961.664,A -85,B 0,C 180,E1 14089.717,E2 14089.717} C_VEL
LIN {X 0,Y 430.032,Z 941.588,A -85,B 0,C 180,E1 14088.72,E2 14088.72} C_VEL
LIN {X 0,Y 432.473,Z 919.159,A -85,B 0,C 180,E1 14087.863,E2 14087.863} C_VEL
LIN {X 0,Y 434.239,Z 897.396,A -85,B 0,C 180,E1 14087.276,E2 14087.276} C_VEL
LIN {X 0,Y 437.332,Z 805.732,A -85,B 0,C 180,E1 14085.648,E2 14085.648} C_VEL
LIN {X 0,Y 443.055,Z 636.442,A -85,B 0,C 180,E1 14082.634,E2 14082.634} C_VEL
LIN {X 0,Y 439.177,Z 614.502,A -85,B 0,C 180,E1 14081.492,E2 14081.492} C_VEL
LIN {X 0,Y 429.764,Z 599.481,A -85,B 0,C 180,E1 14079.517,E2 14079.517} C_VEL
LIN {X 0,Y 425.494,Z 605.291,A -85,B 0,C 180,E1 14078.903,E2 14078.903} C_VEL
LIN {X 0,Y 422.132,Z 608.163,A -85,B 0,C 180,E1 14078.358,E2 14078.358} C_VEL
LIN {X 0,Y 420.675,Z 609.228,A -85,B 0,C 180,E1 14078.112,E2 14078.112} C_VEL
LIN {X 0,Y 416.061,Z 616.571,A -85,B 0,C 180,E1 14077.424,E2 14077.424} C_VEL
LIN {X 0,Y 413.305,Z 619.383,A -85,B 0,C 180,E1 14076.954,E2 14076.954} C_VEL
LIN {X 0,Y 411.53,Z 620.825,A -85,B 0,C 180,E1 14076.531,E2 14076.531} C_VEL
LIN {X 0,Y 410.962,Z 624.281,A -85,B 0,C 180,E1 14076.123,E2 14076.123} C_VEL
LIN {X 0,Y 408.61,Z 668.199,A -85,B 0,C 180,E1 14072.239,E2 14072.239} C_VEL
LIN {X 0,Y 406.248,Z 711.409,A -85,B 0,C 180,E1 14068.441,E2 14068.441} C_VEL
LIN {X 0,Y 405.765,Z 723.559,A -85,B 0,C 180,E1 14067.414,E2 14067.414} C_VEL
LIN {X 0,Y 406.459,Z 732.083,A -85,B 0,C 180,E1 14067.177,E2 14067.177} C_VEL
LIN {X 0,Y 402.534,Z 895.18,A -85,B 0,C 180,E1 14063.84,E2 14063.84} C_VEL
LIN {X 0,Y 402.056,Z 912.896,A -85,B 0,C 180,E1 14063.218,E2 14063.218} C_VEL
LIN {X 0,Y 401.287,Z 930.351,A -85,B 0,C 180,E1 14062.332,E2 14062.332} C_VEL
LIN {X 0,Y 400.359,Z 946.706,A -85,B 0,C 180,E1 14061.231,E2 14061.231} C_VEL
LIN {X 0,Y 399.287,Z 961.984,A -85,B 0,C 180,E1 14059.911,E2 14059.911} C_VEL
LIN {X 0,Y 398.114,Z 976.926,A -85,B 0,C 180,E1 14058.297,E2 14058.297} C_VEL
LIN {X 0,Y 396.996,Z 990.15,A -85,B 0,C 180,E1 14056.535,E2 14056.535} C_VEL
LIN {X 0,Y 395.974,Z 1001.716,A -85,B 0,C 180,E1 14054.626,E2 14054.626} C_VEL
LIN {X 0,Y 395.12,Z 1011.848,A -85,B 0,C 180,E1 14052.57,E2 14052.57} C_VEL
LIN {X 0,Y 394.444,Z 1020.55,A -85,B 0,C 180,E1 14050.369,E2 14050.369} C_VEL
LIN {X 0,Y 393.951,Z 1027.667,A -85,B 0,C 180,E1 14048.025,E2 14048.025} C_VEL
LIN {X 0,Y 393.664,Z 1033.208,A -85,B 0,C 180,E1 14045.539,E2 14045.539} C_VEL
LIN {X 0,Y 393.565,Z 1036.706,A -85,B 0,C 180,E1 14043.204,E2 14043.204} C_VEL
LIN {X 0,Y 393.578,Z 1038.631,A -85,B 0,C 180,E1 14040.728,E2 14040.728} C_VEL
LIN {X 0,Y 393.678,Z 1038.811,A -85,B 0,C 180,E1 14038.254,E2 14038.254} C_VEL
LIN {X 0,Y 393.899,Z 1037.25,A -85,B 0,C 180,E1 14035.779,E2 14035.779} C_VEL
LIN {X 0,Y 394.241,Z 1034.062,A -85,B 0,C 180,E1 14033.447,E2 14033.447} C_VEL
LIN {X 0,Y 394.783,Z 1028.873,A -85,B 0,C 180,E1 14031.023,E2 14031.023} C_VEL
LIN {X 0,Y 395.497,Z 1022.193,A -85,B 0,C 180,E1 14028.775,E2 14028.775} C_VEL
LIN {X 0,Y 396.317,Z 1014.26,A -85,B 0,C 180,E1 14026.728,E2 14026.728} C_VEL
LIN {X 0,Y 397.327,Z 1004.135,A -85,B 0,C 180,E1 14024.679,E2 14024.679} C_VEL
LIN {X 0,Y 398.404,Z 992.826,A -85,B 0,C 180,E1 14022.85,E2 14022.85} C_VEL
LIN {X 0,Y 399.459,Z 980.454,A -85,B 0,C 180,E1 14021.238,E2 14021.238} C_VEL
LIN {X 0,Y 400.46,Z 966.358,A -85,B 0,C 180,E1 14019.77,E2 14019.77} C_VEL
LIN {X 0,Y 401.325,Z 951.195,A -85,B 0,C 180,E1 14018.517,E2 14018.517} C_VEL
LIN {X 0,Y 401.992,Z 935.449,A -85,B 0,C 180,E1 14017.517,E2 14017.517} C_VEL
LIN {X 0,Y 402.464,Z 917.421,A -85,B 0,C 180,E1 14016.681,E2 14016.681} C_VEL
LIN {X 0,Y 402.632,Z 899.573,A -85,B 0,C 180,E1 14016.135,E2 14016.135} C_VEL
LIN {X 0,Y 404.453,Z 823.892,A -85,B 0,C 180,E1 14014.474,E2 14014.474} C_VEL
LIN {X 0,Y 407.838,Z 742.181,A -85,B 0,C 180,E1 14012.516,E2 14012.516} C_VEL
LIN {X 0,Y 409.935,Z 731.757,A -85,B 0,C 180,E1 14011.839,E2 14011.839} C_VEL
LIN {X 0,Y 411.814,Z 688.867,A -85,B 0,C 180,E1 14008.289,E2 14008.289} C_VEL
LIN {X 0,Y 412.648,Z 671.784,A -85,B 0,C 180,E1 14006.881,E2 14006.881} C_VEL
LIN {X 0,Y 413.662,Z 669.627,A -85,B 0,C 180,E1 14006.558,E2 14006.558} C_VEL
LIN {X 0,Y 416.668,Z 666.632,A -85,B 0,C 180,E1 14006.068,E2 14006.068} C_VEL
LIN {X 0,Y 420.817,Z 659.908,A -85,B 0,C 180,E1 14005.503,E2 14005.503} C_VEL
LIN {X 0,Y 422.19,Z 657.625,A -85,B 0,C 180,E1 14005.322,E2 14005.322} C_VEL
LIN {X 0,Y 426.082,Z 653.896,A -85,B 0,C 180,E1 14004.742,E2 14004.742} C_VEL
LIN {X 0,Y 430.307,Z 647.538,A -85,B 0,C 180,E1 14004.196,E2 14004.196} C_VEL
LIN {X 0,Y 431.782,Z 645.165,A -85,B 0,C 180,E1 14004.014,E2 14004.014} C_VEL
LIN {X 0,Y 436.253,Z 640.577,A -85,B 0,C 180,E1 14003.403,E2 14003.403} C_VEL
LIN {X 0,Y 441.393,Z 633.08,A -85,B 0,C 180,E1 14002.785,E2 14002.785} C_VEL
LIN {X 0,Y 446.45,Z 627.67,A -85,B 0,C 180,E1 14002.147,E2 14002.147} C_VEL
LIN {X 0,Y 446.633,Z 627.589,A -85,B 0,C 180,E1 14002.122,E2 14002.122} C_VEL
LIN {X 0,Y 438.205,Z 832.645,A -85,B 0,C 180,E1 13998.228,E2 13998.228} C_VEL
LIN {X 0,Y 435.574,Z 893.986,A -85,B 0,C 180,E1 13997.034,E2 13997.034} C_VEL
LIN {X 0,Y 433.521,Z 917.302,A -85,B 0,C 180,E1 13996.373,E2 13996.373} C_VEL
LIN {X 0,Y 430.837,Z 941.345,A -85,B 0,C 180,E1 13995.436,E2 13995.436} C_VEL
LIN {X 0,Y 428.101,Z 961.468,A -85,B 0,C 180,E1 13994.434,E2 13994.434} C_VEL
LIN {X 0,Y 424.592,Z 983.627,A -85,B 0,C 180,E1 13993.072,E2 13993.072} C_VEL
LIN {X 0,Y 421.067,Z 1003.767,A -85,B 0,C 180,E1 13991.584,E2 13991.584} C_VEL
LIN {X 0,Y 417.158,Z 1023.972,A -85,B 0,C 180,E1 13989.789,E2 13989.789} C_VEL
LIN {X 0,Y 413.227,Z 1043.542,A -85,B 0,C 180,E1 13987.747,E2 13987.747} C_VEL
LIN {X 0,Y 409.544,Z 1061.011,A -85,B 0,C 180,E1 13985.612,E2 13985.612} C_VEL
LIN {X 0,Y 405.831,Z 1078.645,A -85,B 0,C 180,E1 13983.106,E2 13983.106} C_VEL
LIN {X 0,Y 402.507,Z 1094.852,A -85,B 0,C 180,E1 13980.448,E2 13980.448} C_VEL
LIN {X 0,Y 399.651,Z 1109.295,A -85,B 0,C 180,E1 13977.67,E2 13977.67} C_VEL
LIN {X 0,Y 397.188,Z 1122.706,A -85,B 0,C 180,E1 13974.667,E2 13974.667} C_VEL
LIN {X 0,Y 395.413,Z 1133.272,A -85,B 0,C 180,E1 13971.874,E2 13971.874} C_VEL
LIN {X 0,Y 393.862,Z 1143.996,A -85,B 0,C 180,E1 13968.501,E2 13968.501} C_VEL
LIN {X 0,Y 392.939,Z 1151.82,A -85,B 0,C 180,E1 13965.497,E2 13965.497} C_VEL
LIN {X 0,Y 392.334,Z 1158.623,A -85,B 0,C 180,E1 13962.212,E2 13962.212} C_VEL
LIN {X 0,Y 392.065,Z 1163.149,A -85,B 0,C 180,E1 13959.394,E2 13959.394} C_VEL
LIN {X 0,Y 391.93,Z 1166.897,A -85,B 0,C 180,E1 13956.151,E2 13956.151} C_VEL
LIN {X 0,Y 391.893,Z 1168.811,A -85,B 0,C 180,E1 13953.364,E2 13953.364} C_VEL
LIN {X 0,Y 391.892,Z 1169.636,A -85,B 0,C 180,E1 13950.585,E2 13950.585} C_VEL
LIN {X 0,Y 391.905,Z 1169.163,A -85,B 0,C 180,E1 13947.368,E2 13947.368} C_VEL
LIN {X 0,Y 391.917,Z 1167.371,A -85,B 0,C 180,E1 13944.437,E2 13944.437} C_VEL
LIN {X 0,Y 392.029,Z 1164.206,A -85,B 0,C 180,E1 13941.345,E2 13941.345} C_VEL
LIN {X 0,Y 392.285,Z 1159.296,A -85,B 0,C 180,E1 13938.162,E2 13938.162} C_VEL
LIN {X 0,Y 392.829,Z 1152.905,A -85,B 0,C 180,E1 13934.953,E2 13934.953} C_VEL
LIN {X 0,Y 393.772,Z 1144.673,A -85,B 0,C 180,E1 13931.74,E2 13931.74} C_VEL
LIN {X 0,Y 395.162,Z 1135.015,A -85,B 0,C 180,E1 13928.611,E2 13928.611} C_VEL
LIN {X 0,Y 396.999,Z 1123.803,A -85,B 0,C 180,E1 13925.604,E2 13925.604} C_VEL
LIN {X 0,Y 399.429,Z 1110.505,A -85,B 0,C 180,E1 13922.575,E2 13922.575} C_VEL
LIN {X 0,Y 402.162,Z 1096.493,A -85,B 0,C 180,E1 13919.853,E2 13919.853} C_VEL
